REGION Network 7: CY26 interface H-shaftLoadingStopperCylinder4
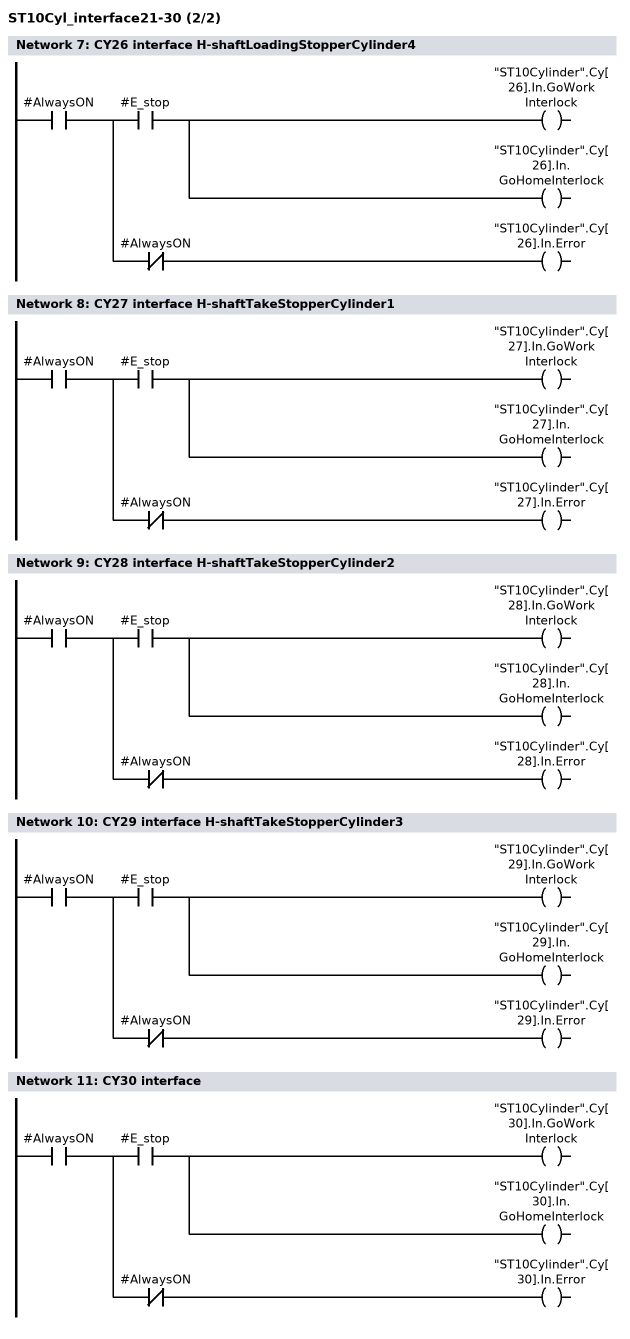
   RUNG wire#powerrail
      Contact( #AlwaysON )
      wire#w1
      Contact( #E_stop )
      wire#w2
      Coil( "ST10Cylinder".Cy[26].In.GoWorkInterlock )
   END_RUNG
   RUNG wire#w2
      Coil( "ST10Cylinder".Cy[26].In.GoHomeInterlock )
   END_RUNG
   RUNG wire#w1
      I_Contact( #AlwaysON )
      Coil( "ST10Cylinder".Cy[26].In.Error )
   END_RUNG
   // the same network as SCL:
   "ST10Cylinder".Cy[26].In.GoWorkInterlock := #AlwaysON AND #E_stop;
   "ST10Cylinder".Cy[26].In.GoHomeInterlock := #AlwaysON AND #E_stop;
   "ST10Cylinder".Cy[26].In.Error := #AlwaysON AND NOT #AlwaysON;
END_REGION

REGION Network 8: CY27 interface H-shaftTakeStopperCylinder1
   RUNG wire#powerrail
      Contact( #AlwaysON )
      wire#w1
      Contact( #E_stop )
      wire#w2
      Coil( "ST10Cylinder".Cy[27].In.GoWorkInterlock )
   END_RUNG
   RUNG wire#w2
      Coil( "ST10Cylinder".Cy[27].In.GoHomeInterlock )
   END_RUNG
   RUNG wire#w1
      I_Contact( #AlwaysON )
      Coil( "ST10Cylinder".Cy[27].In.Error )
   END_RUNG
   // the same network as SCL:
   "ST10Cylinder".Cy[27].In.GoWorkInterlock := #AlwaysON AND #E_stop;
   "ST10Cylinder".Cy[27].In.GoHomeInterlock := #AlwaysON AND #E_stop;
   "ST10Cylinder".Cy[27].In.Error := #AlwaysON AND NOT #AlwaysON;
END_REGION

REGION Network 9: CY28 interface H-shaftTakeStopperCylinder2
   RUNG wire#powerrail
      Contact( #AlwaysON )
      wire#w1
      Contact( #E_stop )
      wire#w2
      Coil( "ST10Cylinder".Cy[28].In.GoWorkInterlock )
   END_RUNG
   RUNG wire#w2
      Coil( "ST10Cylinder".Cy[28].In.GoHomeInterlock )
   END_RUNG
   RUNG wire#w1
      I_Contact( #AlwaysON )
      Coil( "ST10Cylinder".Cy[28].In.Error )
   END_RUNG
   // the same network as SCL:
   "ST10Cylinder".Cy[28].In.GoWorkInterlock := #AlwaysON AND #E_stop;
   "ST10Cylinder".Cy[28].In.GoHomeInterlock := #AlwaysON AND #E_stop;
   "ST10Cylinder".Cy[28].In.Error := #AlwaysON AND NOT #AlwaysON;
END_REGION

REGION Network 10: CY29 interface H-shaftTakeStopperCylinder3
   RUNG wire#powerrail
      Contact( #AlwaysON )
      wire#w1
      Contact( #E_stop )
      wire#w2
      Coil( "ST10Cylinder".Cy[29].In.GoWorkInterlock )
   END_RUNG
   RUNG wire#w2
      Coil( "ST10Cylinder".Cy[29].In.GoHomeInterlock )
   END_RUNG
   RUNG wire#w1
      I_Contact( #AlwaysON )
      Coil( "ST10Cylinder".Cy[29].In.Error )
   END_RUNG
   // the same network as SCL:
   "ST10Cylinder".Cy[29].In.GoWorkInterlock := #AlwaysON AND #E_stop;
   "ST10Cylinder".Cy[29].In.GoHomeInterlock := #AlwaysON AND #E_stop;
   "ST10Cylinder".Cy[29].In.Error := #AlwaysON AND NOT #AlwaysON;
END_REGION

REGION Network 11: CY30 interface
   RUNG wire#powerrail
      Contact( #AlwaysON )
      wire#w1
      Contact( #E_stop )
      wire#w2
      Coil( "ST10Cylinder".Cy[30].In.GoWorkInterlock )
   END_RUNG
   RUNG wire#w2
      Coil( "ST10Cylinder".Cy[30].In.GoHomeInterlock )
   END_RUNG
   RUNG wire#w1
      I_Contact( #AlwaysON )
      Coil( "ST10Cylinder".Cy[30].In.Error )
   END_RUNG
   // the same network as SCL:
   "ST10Cylinder".Cy[30].In.GoWorkInterlock := #AlwaysON AND #E_stop;
   "ST10Cylinder".Cy[30].In.GoHomeInterlock := #AlwaysON AND #E_stop;
   "ST10Cylinder".Cy[30].In.Error := #AlwaysON AND NOT #AlwaysON;
END_REGION
END_FUNCTION

FUNCTION "ST10Cyl_interface31-40" : Void   // FC1023, LAD
{ S7_Optimized_Access := 'FALSE' }
VERSION : 0.1
// stored: AutoNumber false, IsIECCheckEnabled false, SetENOAutomatically false, UDAEnableTagReadback false
   VAR_INPUT
      AlwaysON : Bool;
      E_stop : Bool;
   END_VAR
   VAR_TEMP
      tTest : Bool;
   END_VAR
BEGIN

REGION Network 1 (SCL): Cylinder 31-40 IO Interface (SCL)

   //Cylinder31 IO  J-magnetLiftingLiftingCylinder
   //Input
   "ST10Cylinder".Cy[31].In.WorkPositionSensor := "iJ-magnetLiftingLiftingCylinderInWP";
   "ST10Cylinder".Cy[31].In.HomePositionSensor := "iJ-magnetLiftingLiftingCylinderInHP";
   //Output
   "oJ-magnetLiftingLiftingCylinderToWP" := "ST10Cylinder".Cy[31].Out.GoWorkPosition;
   "oJ-magnetLiftingLiftingCylinderToHP" := "ST10Cylinder".Cy[31].Out.GoHomePosition;

   //Cylinder32 IO  J-magnetLiftingPalletLocationCylinder
   //Input
   "ST10Cylinder".Cy[32].In.WorkPositionSensor := "iJ-magnetLiftingPalletLocationCylinderInWP";
   "ST10Cylinder".Cy[32].In.HomePositionSensor := "iJ-magnetLiftingPalletLocationCylinderInHP";
   //Output
   "oJ-magnetLiftingPalletLocationCylinderToWP" := "ST10Cylinder".Cy[32].Out.GoWorkPosition;
   "oJ-magnetLiftingPalletLocationCylinderToHP" := "ST10Cylinder".Cy[32].Out.GoHomePosition;

   //Cylinder33 IO  J-magnetLoadingStopperCylinder1
   //Input
   "ST10Cylinder".Cy[33].In.WorkPositionSensor := "oJ-magnetLoadingStopperCylinder1_ToWP";
   "ST10Cylinder".Cy[33].In.HomePositionSensor := "oJ-magnetLoadingStopperCylinder1_ToHP";
   //Output
   "oJ-magnetLoadingStopperCylinder1_ToWP" := "ST10Cylinder".Cy[33].Out.GoWorkPosition;
   "oJ-magnetLoadingStopperCylinder1_ToHP" := "ST10Cylinder".Cy[33].Out.GoHomePosition;

   //Cylinder34 IO  J-magnetLoadingStopperCylinder2
   //Input
   "ST10Cylinder".Cy[34].In.WorkPositionSensor := "oJ-magnetLoadingStopperCylinder2_ToWP";
   "ST10Cylinder".Cy[34].In.HomePositionSensor := "oJ-magnetLoadingStopperCylinder2_ToHP";
   //Output
   "oJ-magnetLoadingStopperCylinder2_ToWP" := "ST10Cylinder".Cy[34].Out.GoWorkPosition;
   "oJ-magnetLoadingStopperCylinder2_ToHP" := "ST10Cylinder".Cy[34].Out.GoHomePosition;

   //Cylinder35 IO  J-magnetLoadingStopperCylinder3
   //Input
   "ST10Cylinder".Cy[35].In.WorkPositionSensor := "oJ-magnetLoadingStopperCylinder3_ToWP";
   "ST10Cylinder".Cy[35].In.HomePositionSensor := "oJ-magnetLoadingStopperCylinder3_ToHP";
   //Output
   "oJ-magnetLoadingStopperCylinder3_ToWP" := "ST10Cylinder".Cy[35].Out.GoWorkPosition;
   "oJ-magnetLoadingStopperCylinder3_ToHP" := "ST10Cylinder".Cy[35].Out.GoHomePosition;

   //Cylinder36 J-magnetLoadingStopperCylinder4
   //Input
   "ST10Cylinder".Cy[36].In.WorkPositionSensor := "oJ-magnetLoadingStopperCylinder4_ToWP";
   "ST10Cylinder".Cy[36].In.HomePositionSensor := "oJ-magnetLoadingStopperCylinder4_ToHP";
   //Output
   "oJ-magnetLoadingStopperCylinder4_ToWP" := "ST10Cylinder".Cy[36].Out.GoWorkPosition;
   "oJ-magnetLoadingStopperCylinder4_ToHP" := "ST10Cylinder".Cy[36].Out.GoHomePosition;

   //Cylinder37 J-magnetTakeStopperCylinder1
   //Input
   "ST10Cylinder".Cy[37].In.WorkPositionSensor := "oJ-magnetTakeStopperCylinder1_ToWP";
   "ST10Cylinder".Cy[37].In.HomePositionSensor := "oJ-magnetTakeStopperCylinder1_ToHP";
   //Output
   "oJ-magnetTakeStopperCylinder1_ToWP" := "ST10Cylinder".Cy[37].Out.GoWorkPosition;
   "oJ-magnetTakeStopperCylinder1_ToHP" := "ST10Cylinder".Cy[37].Out.GoHomePosition;

   //Cylinder38 J-magnetTakeStopperCylinder2
   //Input
   "ST10Cylinder".Cy[38].In.WorkPositionSensor := "oJ-magnetTakeStopperCylinder2_ToWP";
   "ST10Cylinder".Cy[38].In.HomePositionSensor := "oJ-magnetTakeStopperCylinder2_ToHP";
   //Output
   "oJ-magnetTakeStopperCylinder2_ToWP" := "ST10Cylinder".Cy[38].Out.GoWorkPosition;
   "oJ-magnetTakeStopperCylinder2_ToHP" := "ST10Cylinder".Cy[38].Out.GoHomePosition;

   //Cylinder39 J-magnetTakeStopperCylinder3
   //Input
   "ST10Cylinder".Cy[39].In.WorkPositionSensor := "oJ-magnetTakeStopperCylinder3_ToWP";
   "ST10Cylinder".Cy[39].In.HomePositionSensor := "oJ-magnetTakeStopperCylinder3_ToHP";
   //Output
   "oJ-magnetTakeStopperCylinder3_ToWP" := "ST10Cylinder".Cy[39].Out.GoWorkPosition;
   "oJ-magnetTakeStopperCylinder3_ToHP" := "ST10Cylinder".Cy[39].Out.GoHomePosition;

   (*
   //Cylinder40 J-magnetLoadingStopperCylinder4_2
   // //Input
   "ST10Cylinder".Cy[40].In.WorkPositionSensor := "oJ-magnetLoadingStopperCylinder4_2";
   "ST10Cylinder".Cy[40].In.HomePositionSensor := NOT "oJ-magnetLoadingStopperCylinder4_2";
   // //Output
   "oJ-magnetLoadingStopperCylinder4_2" := "ST10Cylinder".Cy[40].Out.GoWorkPosition;
   "Feeding washer  lift Cylinder ToHP" := "ST10Cylinder".Cy[40].Out.GoHomePosition;
   *)
END_REGION

REGION Network 2: CY31 interface J-magnetLiftingLiftingCylinder
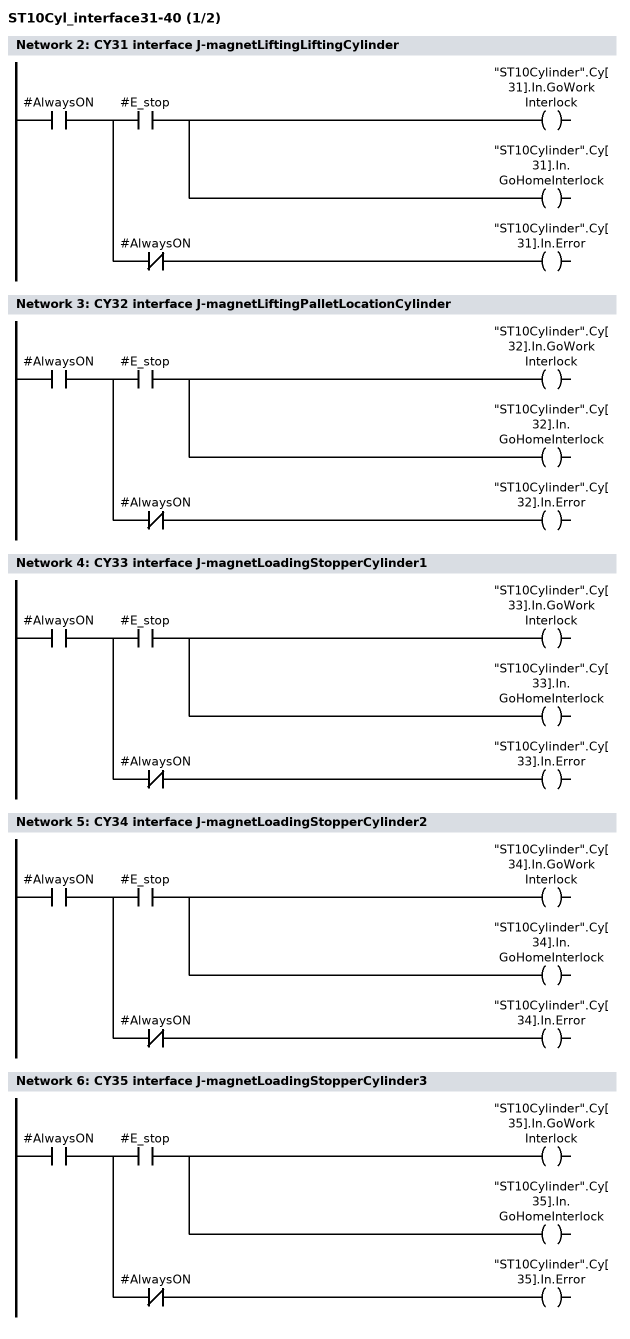
   RUNG wire#powerrail
      Contact( #AlwaysON )
      wire#w1
      Contact( #E_stop )
      wire#w2
      Coil( "ST10Cylinder".Cy[31].In.GoWorkInterlock )
   END_RUNG
   RUNG wire#w2
      Coil( "ST10Cylinder".Cy[31].In.GoHomeInterlock )
   END_RUNG
   RUNG wire#w1
      I_Contact( #AlwaysON )
      Coil( "ST10Cylinder".Cy[31].In.Error )
   END_RUNG
   // the same network as SCL:
   "ST10Cylinder".Cy[31].In.GoWorkInterlock := #AlwaysON AND #E_stop;
   "ST10Cylinder".Cy[31].In.GoHomeInterlock := #AlwaysON AND #E_stop;
   "ST10Cylinder".Cy[31].In.Error := #AlwaysON AND NOT #AlwaysON;
END_REGION

REGION Network 3: CY32 interface J-magnetLiftingPalletLocationCylinder
   RUNG wire#powerrail
      Contact( #AlwaysON )
      wire#w1
      Contact( #E_stop )
      wire#w2
      Coil( "ST10Cylinder".Cy[32].In.GoWorkInterlock )
   END_RUNG
   RUNG wire#w2
      Coil( "ST10Cylinder".Cy[32].In.GoHomeInterlock )
   END_RUNG
   RUNG wire#w1
      I_Contact( #AlwaysON )
      Coil( "ST10Cylinder".Cy[32].In.Error )
   END_RUNG
   // the same network as SCL:
   "ST10Cylinder".Cy[32].In.GoWorkInterlock := #AlwaysON AND #E_stop;
   "ST10Cylinder".Cy[32].In.GoHomeInterlock := #AlwaysON AND #E_stop;
   "ST10Cylinder".Cy[32].In.Error := #AlwaysON AND NOT #AlwaysON;
END_REGION

REGION Network 4: CY33 interface J-magnetLoadingStopperCylinder1
   RUNG wire#powerrail
      Contact( #AlwaysON )
      wire#w1
      Contact( #E_stop )
      wire#w2
      Coil( "ST10Cylinder".Cy[33].In.GoWorkInterlock )
   END_RUNG
   RUNG wire#w2
      Coil( "ST10Cylinder".Cy[33].In.GoHomeInterlock )
   END_RUNG
   RUNG wire#w1
      I_Contact( #AlwaysON )
      Coil( "ST10Cylinder".Cy[33].In.Error )
   END_RUNG
   // the same network as SCL:
   "ST10Cylinder".Cy[33].In.GoWorkInterlock := #AlwaysON AND #E_stop;
   "ST10Cylinder".Cy[33].In.GoHomeInterlock := #AlwaysON AND #E_stop;
   "ST10Cylinder".Cy[33].In.Error := #AlwaysON AND NOT #AlwaysON;
END_REGION

REGION Network 5: CY34 interface J-magnetLoadingStopperCylinder2
   RUNG wire#powerrail
      Contact( #AlwaysON )
      wire#w1
      Contact( #E_stop )
      wire#w2
      Coil( "ST10Cylinder".Cy[34].In.GoWorkInterlock )
   END_RUNG
   RUNG wire#w2
      Coil( "ST10Cylinder".Cy[34].In.GoHomeInterlock )
   END_RUNG
   RUNG wire#w1
      I_Contact( #AlwaysON )
      Coil( "ST10Cylinder".Cy[34].In.Error )
   END_RUNG
   // the same network as SCL:
   "ST10Cylinder".Cy[34].In.GoWorkInterlock := #AlwaysON AND #E_stop;
   "ST10Cylinder".Cy[34].In.GoHomeInterlock := #AlwaysON AND #E_stop;
   "ST10Cylinder".Cy[34].In.Error := #AlwaysON AND NOT #AlwaysON;
END_REGION

REGION Network 6: CY35 interface J-magnetLoadingStopperCylinder3
   RUNG wire#powerrail
      Contact( #AlwaysON )
      wire#w1
      Contact( #E_stop )
      wire#w2
      Coil( "ST10Cylinder".Cy[35].In.GoWorkInterlock )
   END_RUNG
   RUNG wire#w2
      Coil( "ST10Cylinder".Cy[35].In.GoHomeInterlock )
   END_RUNG
   RUNG wire#w1
      I_Contact( #AlwaysON )
      Coil( "ST10Cylinder".Cy[35].In.Error )
   END_RUNG
   // the same network as SCL:
   "ST10Cylinder".Cy[35].In.GoWorkInterlock := #AlwaysON AND #E_stop;
   "ST10Cylinder".Cy[35].In.GoHomeInterlock := #AlwaysON AND #E_stop;
   "ST10Cylinder".Cy[35].In.Error := #AlwaysON AND NOT #AlwaysON;
END_REGION

REGION Network 7: CY36 interface J-magnetLoadingStopperCylinder4
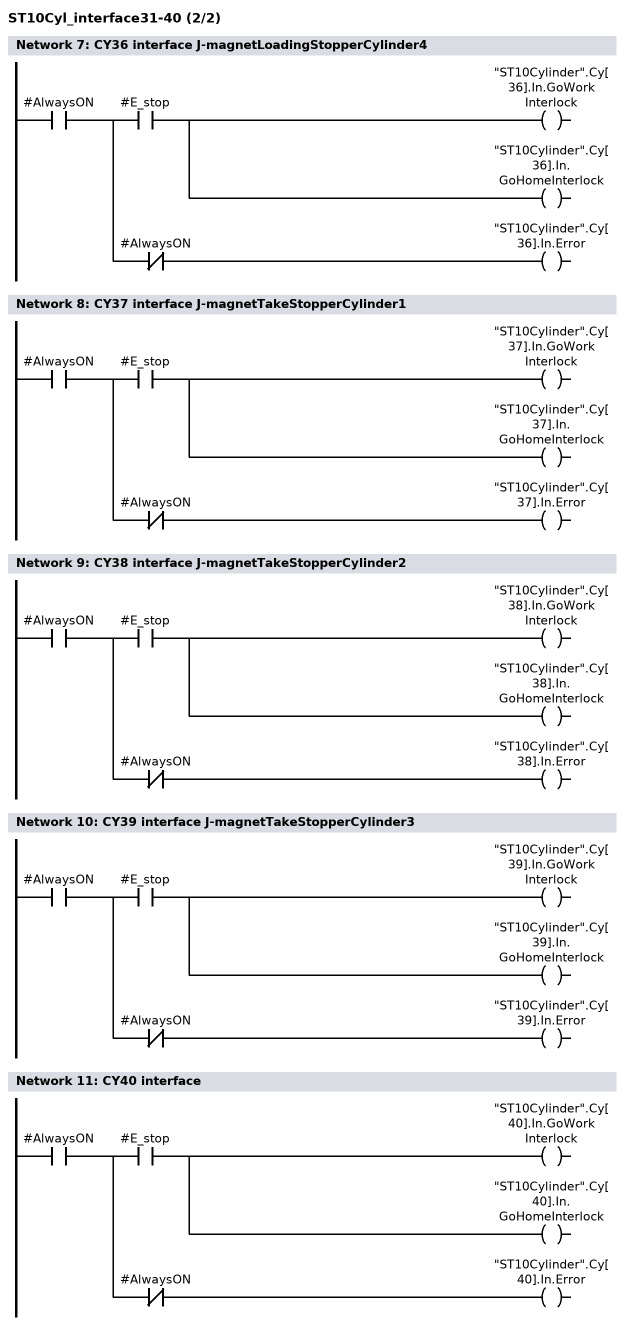
   RUNG wire#powerrail
      Contact( #AlwaysON )
      wire#w1
      Contact( #E_stop )
      wire#w2
      Coil( "ST10Cylinder".Cy[36].In.GoWorkInterlock )
   END_RUNG
   RUNG wire#w2
      Coil( "ST10Cylinder".Cy[36].In.GoHomeInterlock )
   END_RUNG
   RUNG wire#w1
      I_Contact( #AlwaysON )
      Coil( "ST10Cylinder".Cy[36].In.Error )
   END_RUNG
   // the same network as SCL:
   "ST10Cylinder".Cy[36].In.GoWorkInterlock := #AlwaysON AND #E_stop;
   "ST10Cylinder".Cy[36].In.GoHomeInterlock := #AlwaysON AND #E_stop;
   "ST10Cylinder".Cy[36].In.Error := #AlwaysON AND NOT #AlwaysON;
END_REGION

REGION Network 8: CY37 interface J-magnetTakeStopperCylinder1
   RUNG wire#powerrail
      Contact( #AlwaysON )
      wire#w1
      Contact( #E_stop )
      wire#w2
      Coil( "ST10Cylinder".Cy[37].In.GoWorkInterlock )
   END_RUNG
   RUNG wire#w2
      Coil( "ST10Cylinder".Cy[37].In.GoHomeInterlock )
   END_RUNG
   RUNG wire#w1
      I_Contact( #AlwaysON )
      Coil( "ST10Cylinder".Cy[37].In.Error )
   END_RUNG
   // the same network as SCL:
   "ST10Cylinder".Cy[37].In.GoWorkInterlock := #AlwaysON AND #E_stop;
   "ST10Cylinder".Cy[37].In.GoHomeInterlock := #AlwaysON AND #E_stop;
   "ST10Cylinder".Cy[37].In.Error := #AlwaysON AND NOT #AlwaysON;
END_REGION

REGION Network 9: CY38 interface J-magnetTakeStopperCylinder2
   RUNG wire#powerrail
      Contact( #AlwaysON )
      wire#w1
      Contact( #E_stop )
      wire#w2
      Coil( "ST10Cylinder".Cy[38].In.GoWorkInterlock )
   END_RUNG
   RUNG wire#w2
      Coil( "ST10Cylinder".Cy[38].In.GoHomeInterlock )
   END_RUNG
   RUNG wire#w1
      I_Contact( #AlwaysON )
      Coil( "ST10Cylinder".Cy[38].In.Error )
   END_RUNG
   // the same network as SCL:
   "ST10Cylinder".Cy[38].In.GoWorkInterlock := #AlwaysON AND #E_stop;
   "ST10Cylinder".Cy[38].In.GoHomeInterlock := #AlwaysON AND #E_stop;
   "ST10Cylinder".Cy[38].In.Error := #AlwaysON AND NOT #AlwaysON;
END_REGION

REGION Network 10: CY39 interface J-magnetTakeStopperCylinder3
   RUNG wire#powerrail
      Contact( #AlwaysON )
      wire#w1
      Contact( #E_stop )
      wire#w2
      Coil( "ST10Cylinder".Cy[39].In.GoWorkInterlock )
   END_RUNG
   RUNG wire#w2
      Coil( "ST10Cylinder".Cy[39].In.GoHomeInterlock )
   END_RUNG
   RUNG wire#w1
      I_Contact( #AlwaysON )
      Coil( "ST10Cylinder".Cy[39].In.Error )
   END_RUNG
   // the same network as SCL:
   "ST10Cylinder".Cy[39].In.GoWorkInterlock := #AlwaysON AND #E_stop;
   "ST10Cylinder".Cy[39].In.GoHomeInterlock := #AlwaysON AND #E_stop;
   "ST10Cylinder".Cy[39].In.Error := #AlwaysON AND NOT #AlwaysON;
END_REGION

REGION Network 11: CY40 interface
   RUNG wire#powerrail
      Contact( #AlwaysON )
      wire#w1
      Contact( #E_stop )
      wire#w2
      Coil( "ST10Cylinder".Cy[40].In.GoWorkInterlock )
   END_RUNG
   RUNG wire#w2
      Coil( "ST10Cylinder".Cy[40].In.GoHomeInterlock )
   END_RUNG
   RUNG wire#w1
      I_Contact( #AlwaysON )
      Coil( "ST10Cylinder".Cy[40].In.Error )
   END_RUNG
   // the same network as SCL:
   "ST10Cylinder".Cy[40].In.GoWorkInterlock := #AlwaysON AND #E_stop;
   "ST10Cylinder".Cy[40].In.GoHomeInterlock := #AlwaysON AND #E_stop;
   "ST10Cylinder".Cy[40].In.Error := #AlwaysON AND NOT #AlwaysON;
END_REGION
END_FUNCTION

FUNCTION "ST10Cyl_interface41-50" : Void   // FC1024, LAD
{ S7_Optimized_Access := 'FALSE' }
// stored: AutoNumber false, SetENOAutomatically false
   VAR_INPUT
      AlwaysON : Bool;
      E_stop : Bool;
   END_VAR
   VAR_TEMP
      tTest : Bool;
   END_VAR
BEGIN

REGION Network 1 (SCL): Cylinder 41-50 IO Interface (SCL)
   //Cylinder41 IO  K-reserveLifting3LiftingCylinder
   //Input
   "ST10Cylinder".Cy[41].In.WorkPositionSensor := "iK-reserveLifting3LiftingCylinderInWP";
   "ST10Cylinder".Cy[41].In.HomePositionSensor := "iK-reserveLifting3LiftingCylinderInHP";
   //Output
   "oK-reserveLifting3LiftingCylinderToWP" := "ST10Cylinder".Cy[41].Out.GoWorkPosition;
   "oK-reserveLifting3LiftingCylinderToHP" := "ST10Cylinder".Cy[41].Out.GoHomePosition;

   //Cylinder42 IO  K-reserveLifting3PalletLocationCylinder
   //Input
   "ST10Cylinder".Cy[42].In.WorkPositionSensor := "iK-reserveLifting3PalletLocationCylinderInWP";
   "ST10Cylinder".Cy[42].In.HomePositionSensor := "iK-reserveLifting3PalletLocationCylinderInHP";
   //Output
   "oK-reserveLifting3PalletLocationCylinderToWP" := "ST10Cylinder".Cy[42].Out.GoWorkPosition;
   "oK-reserveLifting3PalletLocationCylinderToHP" := "ST10Cylinder".Cy[42].Out.GoHomePosition;

   //Cylinder43 IO  K-reserveLoadingStopperCylinder1
   //Input
   "ST10Cylinder".Cy[43].In.WorkPositionSensor := "oK-reserveLoadingStopperCylinder1_ToWP";
   "ST10Cylinder".Cy[43].In.HomePositionSensor := "oK-reserveLoadingStopperCylinder1_ToHP";
   //Output
   "oK-reserveLoadingStopperCylinder1_ToWP" := "ST10Cylinder".Cy[43].Out.GoWorkPosition;
   "oK-reserveLoadingStopperCylinder1_ToHP" := "ST10Cylinder".Cy[43].Out.GoHomePosition;

   //Cylinder44 IO  K-reserveLoadingStopperCylinder2
   //Input
   "ST10Cylinder".Cy[44].In.WorkPositionSensor := "oK-reserveLoadingStopperCylinder2_ToWP";
   "ST10Cylinder".Cy[44].In.HomePositionSensor := "oK-reserveLoadingStopperCylinder2_ToHP";
   //Output
   "oK-reserveLoadingStopperCylinder2_ToWP" := "ST10Cylinder".Cy[44].Out.GoWorkPosition;
   "oK-reserveLoadingStopperCylinder2_ToHP" := "ST10Cylinder".Cy[44].Out.GoHomePosition;

   //Cylinder45 IO  K-reserveLoadingStopperCylinder3
   //Input
   "ST10Cylinder".Cy[45].In.WorkPositionSensor := "oK-reserveLoadingStopperCylinder3_ToWP";
   "ST10Cylinder".Cy[45].In.HomePositionSensor := "oK-reserveLoadingStopperCylinder3_ToHP";
   //Output
   "oK-reserveLoadingStopperCylinder3_ToWP" := "ST10Cylinder".Cy[45].Out.GoWorkPosition;
   "oK-reserveLoadingStopperCylinder3_ToHP" := "ST10Cylinder".Cy[45].Out.GoHomePosition;

   //Cylinder46 K-reserveLoadingStopperCylinder4
   //Input
   "ST10Cylinder".Cy[46].In.WorkPositionSensor := "oK-reserveLoadingStopperCylinder4_ToWP";
   "ST10Cylinder".Cy[46].In.HomePositionSensor := "oK-reserveLoadingStopperCylinder4_ToHP";
   //Output
   "oK-reserveLoadingStopperCylinder4_ToWP" := "ST10Cylinder".Cy[46].Out.GoWorkPosition;
   "oK-reserveLoadingStopperCylinder4_ToHP" := "ST10Cylinder".Cy[46].Out.GoHomePosition;

   //Cylinder47 K-reserveTakeStopperCylinder1
   //Input
   "ST10Cylinder".Cy[47].In.WorkPositionSensor := "oK-reserveTakeStopperCylinder1_ToWP";
   "ST10Cylinder".Cy[47].In.HomePositionSensor := "oK-reserveTakeStopperCylinder1_ToHP";
   //Output
   "oK-reserveTakeStopperCylinder1_ToWP" := "ST10Cylinder".Cy[47].Out.GoWorkPosition;
   "oK-reserveTakeStopperCylinder1_ToHP" := "ST10Cylinder".Cy[47].Out.GoHomePosition;

   //Cylinder48 K-reserveTakeStopperCylinder2
   //Input
   "ST10Cylinder".Cy[48].In.WorkPositionSensor := "oK-reserveTakeStopperCylinder2_ToWP";
   "ST10Cylinder".Cy[48].In.HomePositionSensor := "oK-reserveTakeStopperCylinder2_ToHP";
   //Output
   "oK-reserveTakeStopperCylinder2_ToWP" := "ST10Cylinder".Cy[48].Out.GoWorkPosition;
   "oK-reserveTakeStopperCylinder2_ToHP" := "ST10Cylinder".Cy[48].Out.GoHomePosition;

   //Cylinder49 K-reserveTakeStopperCylinder3
   //Input
   "ST10Cylinder".Cy[49].In.WorkPositionSensor := "oK-reserveTakeStopperCylinder3_ToWP";
   "ST10Cylinder".Cy[49].In.HomePositionSensor := "oK-reserveTakeStopperCylinder3_ToHP";
   //Output
   "oK-reserveTakeStopperCylinder3_ToWP" := "ST10Cylinder".Cy[49].Out.GoWorkPosition;
   "oK-reserveTakeStopperCylinder3_ToHP" := "ST10Cylinder".Cy[49].Out.GoHomePosition;

   (*
   //Cylinder50 K-reserveLoadingStopperCylinder4_2
   // //Input
   "ST10Cylinder".Cy[50].In.WorkPositionSensor := "oK-reserveLoadingStopperCylinder4_2";
   "ST10Cylinder".Cy[50].In.HomePositionSensor := NOT "oK-reserveLoadingStopperCylinder4_2";
   // //Output
   "oK-reserveLoadingStopperCylinder4_2" := "ST10Cylinder".Cy[50].Out.GoWorkPosition;
   // "Feeding washer  lift Cylinder ToHP" := "ST10Cylinder".Cy[50].Out.GoHomePosition;
   *)
END_REGION

REGION Network 2: CY41 interface K-reserveLifting3LiftingCylinder
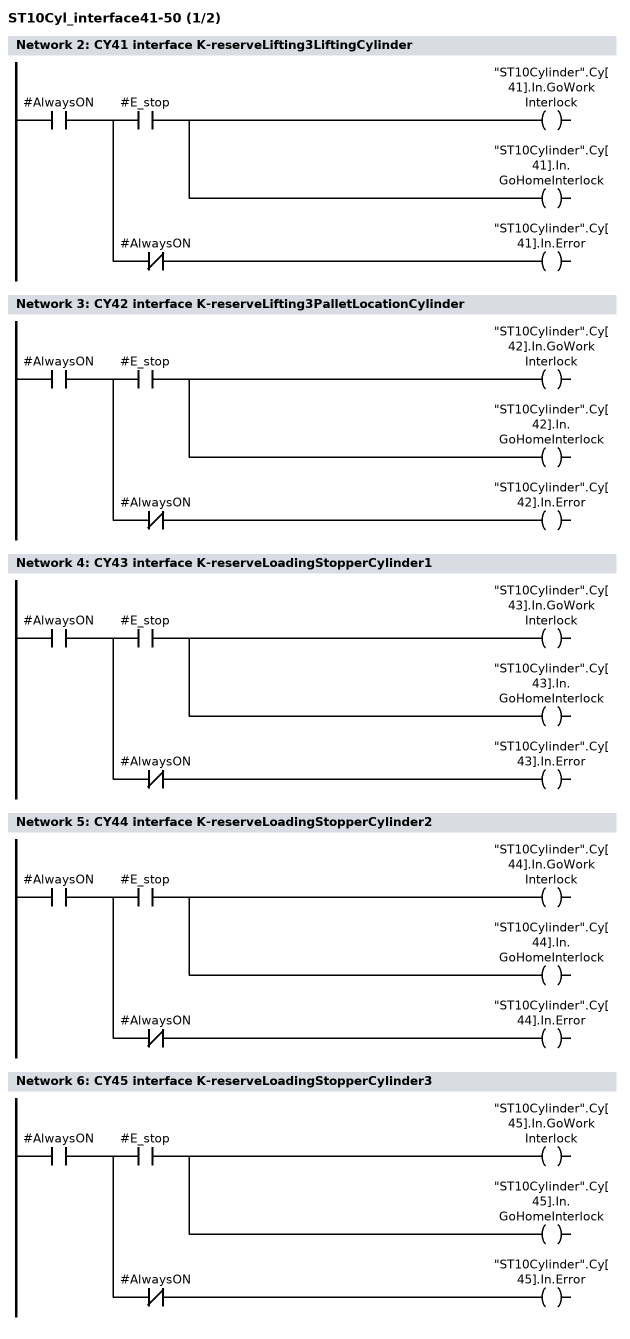
   RUNG wire#powerrail
      Contact( #AlwaysON )
      wire#w1
      Contact( #E_stop )
      wire#w2
      Coil( "ST10Cylinder".Cy[41].In.GoWorkInterlock )
   END_RUNG
   RUNG wire#w2
      Coil( "ST10Cylinder".Cy[41].In.GoHomeInterlock )
   END_RUNG
   RUNG wire#w1
      I_Contact( #AlwaysON )
      Coil( "ST10Cylinder".Cy[41].In.Error )
   END_RUNG
   // the same network as SCL:
   "ST10Cylinder".Cy[41].In.GoWorkInterlock := #AlwaysON AND #E_stop;
   "ST10Cylinder".Cy[41].In.GoHomeInterlock := #AlwaysON AND #E_stop;
   "ST10Cylinder".Cy[41].In.Error := #AlwaysON AND NOT #AlwaysON;
END_REGION

REGION Network 3: CY42 interface K-reserveLifting3PalletLocationCylinder
   RUNG wire#powerrail
      Contact( #AlwaysON )
      wire#w1
      Contact( #E_stop )
      wire#w2
      Coil( "ST10Cylinder".Cy[42].In.GoWorkInterlock )
   END_RUNG
   RUNG wire#w2
      Coil( "ST10Cylinder".Cy[42].In.GoHomeInterlock )
   END_RUNG
   RUNG wire#w1
      I_Contact( #AlwaysON )
      Coil( "ST10Cylinder".Cy[42].In.Error )
   END_RUNG
   // the same network as SCL:
   "ST10Cylinder".Cy[42].In.GoWorkInterlock := #AlwaysON AND #E_stop;
   "ST10Cylinder".Cy[42].In.GoHomeInterlock := #AlwaysON AND #E_stop;
   "ST10Cylinder".Cy[42].In.Error := #AlwaysON AND NOT #AlwaysON;
END_REGION

REGION Network 4: CY43 interface K-reserveLoadingStopperCylinder1
   RUNG wire#powerrail
      Contact( #AlwaysON )
      wire#w1
      Contact( #E_stop )
      wire#w2
      Coil( "ST10Cylinder".Cy[43].In.GoWorkInterlock )
   END_RUNG
   RUNG wire#w2
      Coil( "ST10Cylinder".Cy[43].In.GoHomeInterlock )
   END_RUNG
   RUNG wire#w1
      I_Contact( #AlwaysON )
      Coil( "ST10Cylinder".Cy[43].In.Error )
   END_RUNG
   // the same network as SCL:
   "ST10Cylinder".Cy[43].In.GoWorkInterlock := #AlwaysON AND #E_stop;
   "ST10Cylinder".Cy[43].In.GoHomeInterlock := #AlwaysON AND #E_stop;
   "ST10Cylinder".Cy[43].In.Error := #AlwaysON AND NOT #AlwaysON;
END_REGION

REGION Network 5: CY44 interface K-reserveLoadingStopperCylinder2
   RUNG wire#powerrail
      Contact( #AlwaysON )
      wire#w1
      Contact( #E_stop )
      wire#w2
      Coil( "ST10Cylinder".Cy[44].In.GoWorkInterlock )
   END_RUNG
   RUNG wire#w2
      Coil( "ST10Cylinder".Cy[44].In.GoHomeInterlock )
   END_RUNG
   RUNG wire#w1
      I_Contact( #AlwaysON )
      Coil( "ST10Cylinder".Cy[44].In.Error )
   END_RUNG
   // the same network as SCL:
   "ST10Cylinder".Cy[44].In.GoWorkInterlock := #AlwaysON AND #E_stop;
   "ST10Cylinder".Cy[44].In.GoHomeInterlock := #AlwaysON AND #E_stop;
   "ST10Cylinder".Cy[44].In.Error := #AlwaysON AND NOT #AlwaysON;
END_REGION

REGION Network 6: CY45 interface K-reserveLoadingStopperCylinder3
   RUNG wire#powerrail
      Contact( #AlwaysON )
      wire#w1
      Contact( #E_stop )
      wire#w2
      Coil( "ST10Cylinder".Cy[45].In.GoWorkInterlock )
   END_RUNG
   RUNG wire#w2
      Coil( "ST10Cylinder".Cy[45].In.GoHomeInterlock )
   END_RUNG
   RUNG wire#w1
      I_Contact( #AlwaysON )
      Coil( "ST10Cylinder".Cy[45].In.Error )
   END_RUNG
   // the same network as SCL:
   "ST10Cylinder".Cy[45].In.GoWorkInterlock := #AlwaysON AND #E_stop;
   "ST10Cylinder".Cy[45].In.GoHomeInterlock := #AlwaysON AND #E_stop;
   "ST10Cylinder".Cy[45].In.Error := #AlwaysON AND NOT #AlwaysON;
END_REGION

REGION Network 7: CY46 interface K-reserveLoadingStopperCylinder4
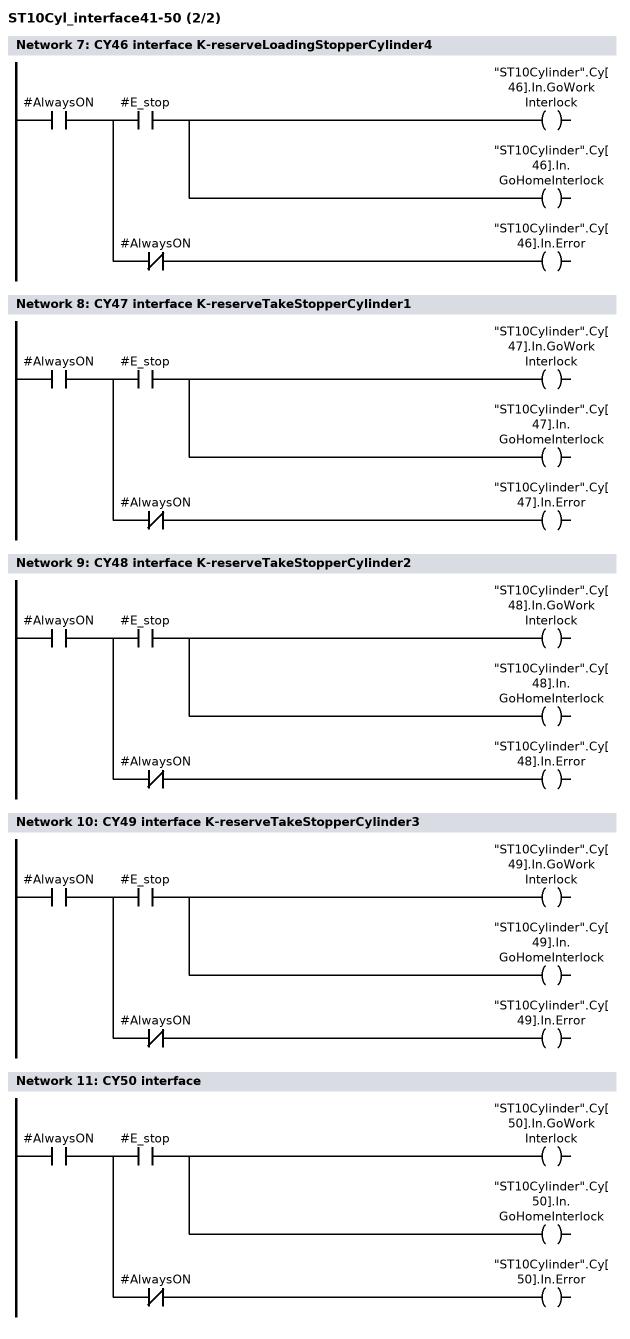
   RUNG wire#powerrail
      Contact( #AlwaysON )
      wire#w1
      Contact( #E_stop )
      wire#w2
      Coil( "ST10Cylinder".Cy[46].In.GoWorkInterlock )
   END_RUNG
   RUNG wire#w2
      Coil( "ST10Cylinder".Cy[46].In.GoHomeInterlock )
   END_RUNG
   RUNG wire#w1
      I_Contact( #AlwaysON )
      Coil( "ST10Cylinder".Cy[46].In.Error )
   END_RUNG
   // the same network as SCL:
   "ST10Cylinder".Cy[46].In.GoWorkInterlock := #AlwaysON AND #E_stop;
   "ST10Cylinder".Cy[46].In.GoHomeInterlock := #AlwaysON AND #E_stop;
   "ST10Cylinder".Cy[46].In.Error := #AlwaysON AND NOT #AlwaysON;
END_REGION

REGION Network 8: CY47 interface K-reserveTakeStopperCylinder1
   RUNG wire#powerrail
      Contact( #AlwaysON )
      wire#w1
      Contact( #E_stop )
      wire#w2
      Coil( "ST10Cylinder".Cy[47].In.GoWorkInterlock )
   END_RUNG
   RUNG wire#w2
      Coil( "ST10Cylinder".Cy[47].In.GoHomeInterlock )
   END_RUNG
   RUNG wire#w1
      I_Contact( #AlwaysON )
      Coil( "ST10Cylinder".Cy[47].In.Error )
   END_RUNG
   // the same network as SCL:
   "ST10Cylinder".Cy[47].In.GoWorkInterlock := #AlwaysON AND #E_stop;
   "ST10Cylinder".Cy[47].In.GoHomeInterlock := #AlwaysON AND #E_stop;
   "ST10Cylinder".Cy[47].In.Error := #AlwaysON AND NOT #AlwaysON;
END_REGION

REGION Network 9: CY48 interface K-reserveTakeStopperCylinder2
   RUNG wire#powerrail
      Contact( #AlwaysON )
      wire#w1
      Contact( #E_stop )
      wire#w2
      Coil( "ST10Cylinder".Cy[48].In.GoWorkInterlock )
   END_RUNG
   RUNG wire#w2
      Coil( "ST10Cylinder".Cy[48].In.GoHomeInterlock )
   END_RUNG
   RUNG wire#w1
      I_Contact( #AlwaysON )
      Coil( "ST10Cylinder".Cy[48].In.Error )
   END_RUNG
   // the same network as SCL:
   "ST10Cylinder".Cy[48].In.GoWorkInterlock := #AlwaysON AND #E_stop;
   "ST10Cylinder".Cy[48].In.GoHomeInterlock := #AlwaysON AND #E_stop;
   "ST10Cylinder".Cy[48].In.Error := #AlwaysON AND NOT #AlwaysON;
END_REGION

REGION Network 10: CY49 interface K-reserveTakeStopperCylinder3
   RUNG wire#powerrail
      Contact( #AlwaysON )
      wire#w1
      Contact( #E_stop )
      wire#w2
      Coil( "ST10Cylinder".Cy[49].In.GoWorkInterlock )
   END_RUNG
   RUNG wire#w2
      Coil( "ST10Cylinder".Cy[49].In.GoHomeInterlock )
   END_RUNG
   RUNG wire#w1
      I_Contact( #AlwaysON )
      Coil( "ST10Cylinder".Cy[49].In.Error )
   END_RUNG
   // the same network as SCL:
   "ST10Cylinder".Cy[49].In.GoWorkInterlock := #AlwaysON AND #E_stop;
   "ST10Cylinder".Cy[49].In.GoHomeInterlock := #AlwaysON AND #E_stop;
   "ST10Cylinder".Cy[49].In.Error := #AlwaysON AND NOT #AlwaysON;
END_REGION

REGION Network 11: CY50 interface
   RUNG wire#powerrail
      Contact( #AlwaysON )
      wire#w1
      Contact( #E_stop )
      wire#w2
      Coil( "ST10Cylinder".Cy[50].In.GoWorkInterlock )
   END_RUNG
   RUNG wire#w2
      Coil( "ST10Cylinder".Cy[50].In.GoHomeInterlock )
   END_RUNG
   RUNG wire#w1
      I_Contact( #AlwaysON )
      Coil( "ST10Cylinder".Cy[50].In.Error )
   END_RUNG
   // the same network as SCL:
   "ST10Cylinder".Cy[50].In.GoWorkInterlock := #AlwaysON AND #E_stop;
   "ST10Cylinder".Cy[50].In.GoHomeInterlock := #AlwaysON AND #E_stop;
   "ST10Cylinder".Cy[50].In.Error := #AlwaysON AND NOT #AlwaysON;
END_REGION
END_FUNCTION

FUNCTION "ST10Cyl_interface51-60" : Void   // FC1025, LAD
{ S7_Optimized_Access := 'FALSE' }
VERSION : 0.1
// stored: AutoNumber false, IsIECCheckEnabled false, SetENOAutomatically false, UDAEnableTagReadback false
   VAR_INPUT
      AlwaysON : Bool;
      E_stop : Bool;
   END_VAR
   VAR_TEMP
      tTest : Bool;
   END_VAR
   VAR_TEMP   // added for the SCL form of the ladder/FBD networks
      _w1 : Bool;
   END_VAR
BEGIN

REGION Network 1 (SCL): Cylinder 51-60 IO Interface (SCL)

   //Cylinder51 IO  L-UnloadingTransCylinder
   //Input
   "ST10Cylinder".Cy[51].In.WorkPositionSensor := "iL-UnloadingTransCylinderInWP";
   "ST10Cylinder".Cy[51].In.HomePositionSensor := "iL-UnloadingTransCylinderInHP";
   //Output
   "oL-UnloadingTransCylinderToWP" := "ST10Cylinder".Cy[51].Out.GoWorkPosition;
   "oL-UnloadingTransCylinderToHP" := "ST10Cylinder".Cy[51].Out.GoHomePosition;

   //Cylinder52 IO  L-UnloadingTransPalletLocationCylinder
   //Input
   "ST10Cylinder".Cy[52].In.WorkPositionSensor := "iL-UnloadingTransPalletLocationCylinderInWP";
   "ST10Cylinder".Cy[52].In.HomePositionSensor := "iL-UnloadingTransPalletLocationCylinderInHP";
   //Output
   "oL-UnloadingTransPalletLocationCylinderToWP" := "ST10Cylinder".Cy[52].Out.GoWorkPosition;
   "oL-UnloadingTransPalletLocationCylinderToHP" := "ST10Cylinder".Cy[52].Out.GoHomePosition;

   //Cylinder53 IO  L-UnloadingStopperCylinder1
   //Input
   "ST10Cylinder".Cy[53].In.WorkPositionSensor := "oL-UnloadingStopperCylinder1_ToWP";
   "ST10Cylinder".Cy[53].In.HomePositionSensor := "oL-UnloadingStopperCylinder1_ToHP";
   //Output
   "oL-UnloadingStopperCylinder1_ToWP" := "ST10Cylinder".Cy[53].Out.GoWorkPosition;
   "oL-UnloadingStopperCylinder1_ToHP" := "ST10Cylinder".Cy[53].Out.GoHomePosition;

   //Cylinder54 IO  L-UnloadingStopperCylinder2
   //Input
   "ST10Cylinder".Cy[54].In.WorkPositionSensor := "oL-UnloadingStopperCylinder2_ToWP";
   "ST10Cylinder".Cy[54].In.HomePositionSensor := "oL-UnloadingStopperCylinder2_ToHP";
   //Output
   "oL-UnloadingStopperCylinder2_ToWP" := "ST10Cylinder".Cy[54].Out.GoWorkPosition;
   "oL-UnloadingStopperCylinder2_ToHP" := "ST10Cylinder".Cy[54].Out.GoHomePosition;

   //Cylinder55 IO  L-UnloadingStopperCylinder3
   //Input
   "ST10Cylinder".Cy[55].In.WorkPositionSensor := "oL-UnloadingStopperCylinder3_ToWP";
   "ST10Cylinder".Cy[55].In.HomePositionSensor := "oL-UnloadingStopperCylinder3_ToHP";
   //Output
   "oL-UnloadingStopperCylinder3_ToWP" := "ST10Cylinder".Cy[55].Out.GoWorkPosition;
   "oL-UnloadingStopperCylinder3_ToHP" := "ST10Cylinder".Cy[55].Out.GoHomePosition;

   (*
   //Cylinder56  L-UnloadingStopperCylinder2_2
   //Input
   "ST10Cylinder".Cy[56].In.WorkPositionSensor := "oL-UnloadingStopperCylinder2_2";
   "ST10Cylinder".Cy[56].In.HomePositionSensor := NOT "oL-UnloadingStopperCylinder2_2";
   //Output
   "oL-UnloadingStopperCylinder2_2" := "ST10Cylinder".Cy[56].Out.GoWorkPosition;
   //"oI-0080TrayLoadingTraySupportCylinder1ToHP" := "ST10Cylinder".Cy[56].Out.GoHomePosition;

   //Cylinder57 L-UnloadingStopperCylinder3_1
   //Input
   "ST10Cylinder".Cy[57].In.WorkPositionSensor := "oL-UnloadingStopperCylinder3_1";
   "ST10Cylinder".Cy[57].In.HomePositionSensor := NOT "oL-UnloadingStopperCylinder3_1";
   //Output
   "oL-UnloadingStopperCylinder3_1" := "ST10Cylinder".Cy[57].Out.GoWorkPosition;
   //"oI-0070TrayLoadingTraySupportCylinder8ToHP" := "ST10Cylinder".Cy[57].Out.GoHomePosition;

   //Cylinder58 L-UnloadingStopperCylinder3_2
   //Input
   "ST10Cylinder".Cy[58].In.WorkPositionSensor := "oL-UnloadingStopperCylinder3_2";
   "ST10Cylinder".Cy[58].In.HomePositionSensor := NOT "oL-UnloadingStopperCylinder3_2";
   //Output
   "oL-UnloadingStopperCylinder3_2" := "ST10Cylinder".Cy[58].Out.GoWorkPosition;
   //"oI-0080TrayLoadingTrayLocationCylinderToHP" := "ST10Cylinder".Cy[58].Out.GoHomePosition;
   //

   *)
END_REGION

REGION Network 2: CY51 interface L-UnloadingTransCylinder
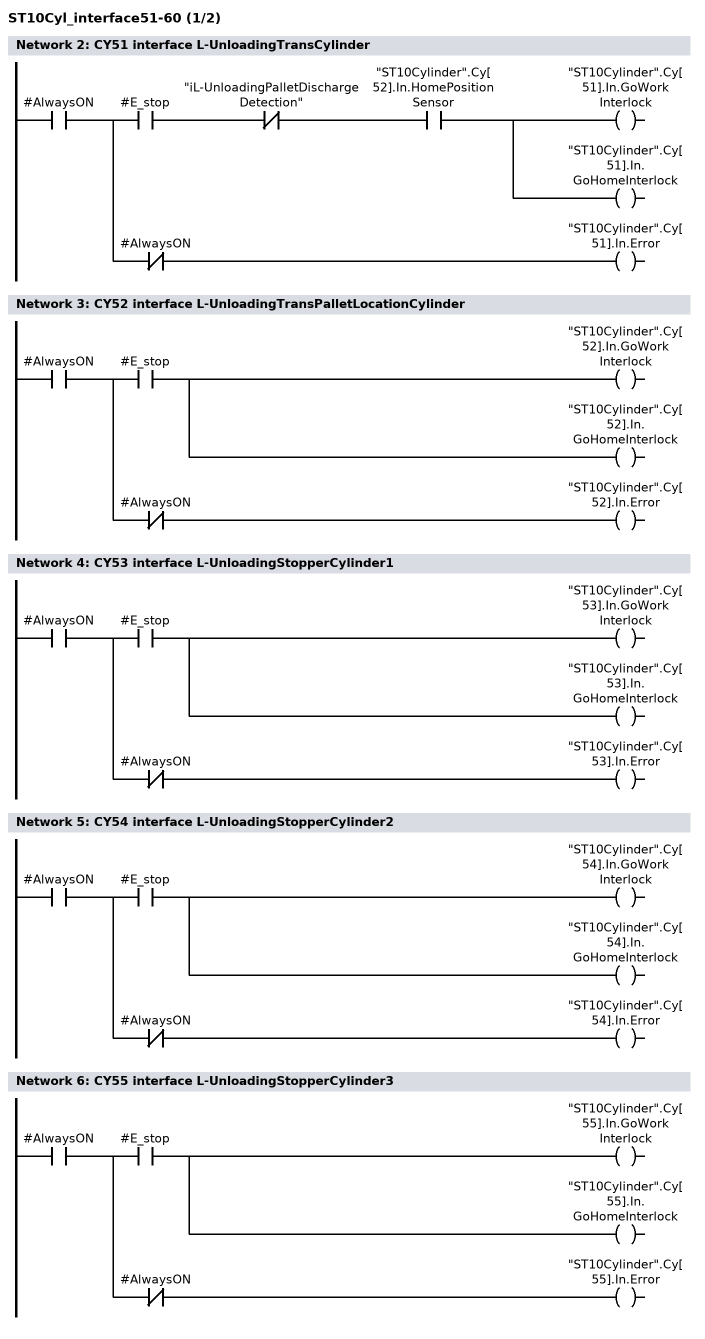
   RUNG wire#powerrail
      Contact( #AlwaysON )
      wire#w1
      Contact( #E_stop )
      I_Contact( "iL-UnloadingPalletDischargeDetection" )
      Contact( "ST10Cylinder".Cy[52].In.HomePositionSensor )
      wire#w2
      Coil( "ST10Cylinder".Cy[51].In.GoWorkInterlock )
   END_RUNG
   RUNG wire#w2
      Coil( "ST10Cylinder".Cy[51].In.GoHomeInterlock )
   END_RUNG
   RUNG wire#w1
      I_Contact( #AlwaysON )
      Coil( "ST10Cylinder".Cy[51].In.Error )
   END_RUNG
   // the same network as SCL:
   #_w1 := #AlwaysON AND #E_stop AND NOT "iL-UnloadingPalletDischargeDetection" AND "ST10Cylinder".Cy[52].In.HomePositionSensor;
   "ST10Cylinder".Cy[51].In.GoWorkInterlock := #AlwaysON AND #E_stop AND NOT "iL-UnloadingPalletDischargeDetection" AND "ST10Cylinder".Cy[52].In.HomePositionSensor;
   "ST10Cylinder".Cy[51].In.GoHomeInterlock := #_w1;
   "ST10Cylinder".Cy[51].In.Error := #AlwaysON AND NOT #AlwaysON;
END_REGION

REGION Network 3: CY52 interface L-UnloadingTransPalletLocationCylinder
   RUNG wire#powerrail
      Contact( #AlwaysON )
      wire#w1
      Contact( #E_stop )
      wire#w2
      Coil( "ST10Cylinder".Cy[52].In.GoWorkInterlock )
   END_RUNG
   RUNG wire#w2
      Coil( "ST10Cylinder".Cy[52].In.GoHomeInterlock )
   END_RUNG
   RUNG wire#w1
      I_Contact( #AlwaysON )
      Coil( "ST10Cylinder".Cy[52].In.Error )
   END_RUNG
   // the same network as SCL:
   "ST10Cylinder".Cy[52].In.GoWorkInterlock := #AlwaysON AND #E_stop;
   "ST10Cylinder".Cy[52].In.GoHomeInterlock := #AlwaysON AND #E_stop;
   "ST10Cylinder".Cy[52].In.Error := #AlwaysON AND NOT #AlwaysON;
END_REGION

REGION Network 4: CY53 interface L-UnloadingStopperCylinder1
   RUNG wire#powerrail
      Contact( #AlwaysON )
      wire#w1
      Contact( #E_stop )
      wire#w2
      Coil( "ST10Cylinder".Cy[53].In.GoWorkInterlock )
   END_RUNG
   RUNG wire#w2
      Coil( "ST10Cylinder".Cy[53].In.GoHomeInterlock )
   END_RUNG
   RUNG wire#w1
      I_Contact( #AlwaysON )
      Coil( "ST10Cylinder".Cy[53].In.Error )
   END_RUNG
   // the same network as SCL:
   "ST10Cylinder".Cy[53].In.GoWorkInterlock := #AlwaysON AND #E_stop;
   "ST10Cylinder".Cy[53].In.GoHomeInterlock := #AlwaysON AND #E_stop;
   "ST10Cylinder".Cy[53].In.Error := #AlwaysON AND NOT #AlwaysON;
END_REGION

REGION Network 5: CY54 interface L-UnloadingStopperCylinder2
   RUNG wire#powerrail
      Contact( #AlwaysON )
      wire#w1
      Contact( #E_stop )
      wire#w2
      Coil( "ST10Cylinder".Cy[54].In.GoWorkInterlock )
   END_RUNG
   RUNG wire#w2
      Coil( "ST10Cylinder".Cy[54].In.GoHomeInterlock )
   END_RUNG
   RUNG wire#w1
      I_Contact( #AlwaysON )
      Coil( "ST10Cylinder".Cy[54].In.Error )
   END_RUNG
   // the same network as SCL:
   "ST10Cylinder".Cy[54].In.GoWorkInterlock := #AlwaysON AND #E_stop;
   "ST10Cylinder".Cy[54].In.GoHomeInterlock := #AlwaysON AND #E_stop;
   "ST10Cylinder".Cy[54].In.Error := #AlwaysON AND NOT #AlwaysON;
END_REGION

REGION Network 6: CY55 interface L-UnloadingStopperCylinder3
   RUNG wire#powerrail
      Contact( #AlwaysON )
      wire#w1
      Contact( #E_stop )
      wire#w2
      Coil( "ST10Cylinder".Cy[55].In.GoWorkInterlock )
   END_RUNG
   RUNG wire#w2
      Coil( "ST10Cylinder".Cy[55].In.GoHomeInterlock )
   END_RUNG
   RUNG wire#w1
      I_Contact( #AlwaysON )
      Coil( "ST10Cylinder".Cy[55].In.Error )
   END_RUNG
   // the same network as SCL:
   "ST10Cylinder".Cy[55].In.GoWorkInterlock := #AlwaysON AND #E_stop;
   "ST10Cylinder".Cy[55].In.GoHomeInterlock := #AlwaysON AND #E_stop;
   "ST10Cylinder".Cy[55].In.Error := #AlwaysON AND NOT #AlwaysON;
END_REGION

REGION Network 7: CY56 interface
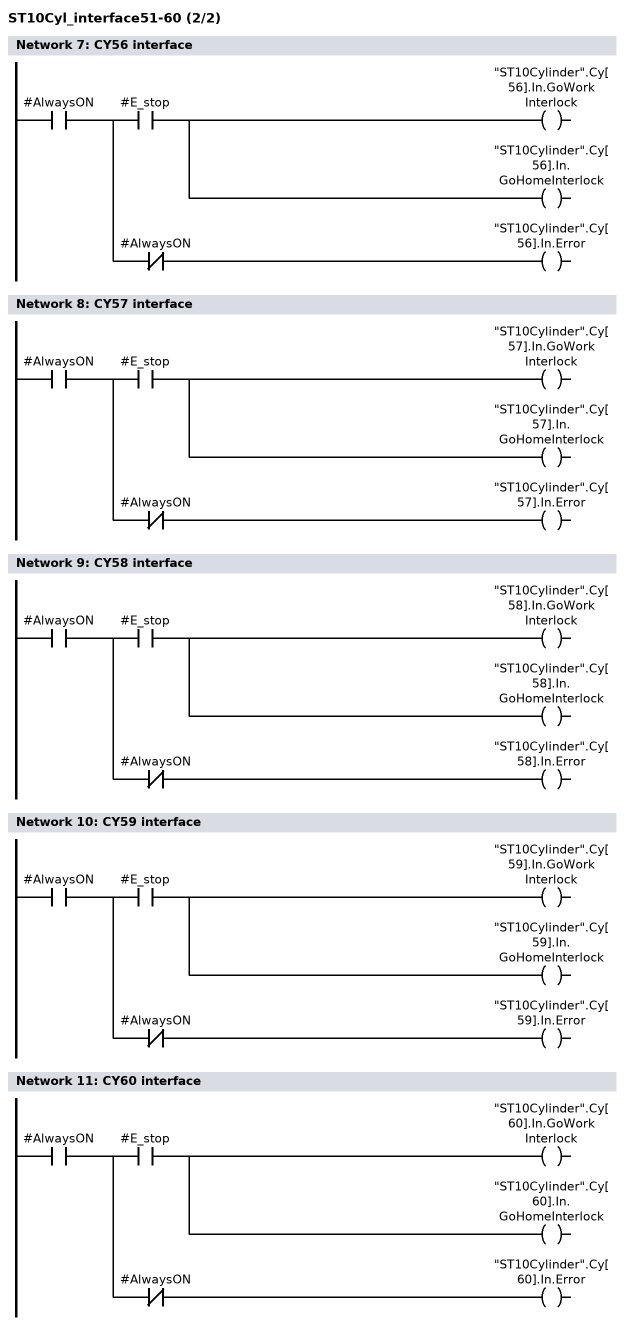
   RUNG wire#powerrail
      Contact( #AlwaysON )
      wire#w1
      Contact( #E_stop )
      wire#w2
      Coil( "ST10Cylinder".Cy[56].In.GoWorkInterlock )
   END_RUNG
   RUNG wire#w2
      Coil( "ST10Cylinder".Cy[56].In.GoHomeInterlock )
   END_RUNG
   RUNG wire#w1
      I_Contact( #AlwaysON )
      Coil( "ST10Cylinder".Cy[56].In.Error )
   END_RUNG
   // the same network as SCL:
   "ST10Cylinder".Cy[56].In.GoWorkInterlock := #AlwaysON AND #E_stop;
   "ST10Cylinder".Cy[56].In.GoHomeInterlock := #AlwaysON AND #E_stop;
   "ST10Cylinder".Cy[56].In.Error := #AlwaysON AND NOT #AlwaysON;
END_REGION

REGION Network 8: CY57 interface
   RUNG wire#powerrail
      Contact( #AlwaysON )
      wire#w1
      Contact( #E_stop )
      wire#w2
      Coil( "ST10Cylinder".Cy[57].In.GoWorkInterlock )
   END_RUNG
   RUNG wire#w2
      Coil( "ST10Cylinder".Cy[57].In.GoHomeInterlock )
   END_RUNG
   RUNG wire#w1
      I_Contact( #AlwaysON )
      Coil( "ST10Cylinder".Cy[57].In.Error )
   END_RUNG
   // the same network as SCL:
   "ST10Cylinder".Cy[57].In.GoWorkInterlock := #AlwaysON AND #E_stop;
   "ST10Cylinder".Cy[57].In.GoHomeInterlock := #AlwaysON AND #E_stop;
   "ST10Cylinder".Cy[57].In.Error := #AlwaysON AND NOT #AlwaysON;
END_REGION

REGION Network 9: CY58 interface
   RUNG wire#powerrail
      Contact( #AlwaysON )
      wire#w1
      Contact( #E_stop )
      wire#w2
      Coil( "ST10Cylinder".Cy[58].In.GoWorkInterlock )
   END_RUNG
   RUNG wire#w2
      Coil( "ST10Cylinder".Cy[58].In.GoHomeInterlock )
   END_RUNG
   RUNG wire#w1
      I_Contact( #AlwaysON )
      Coil( "ST10Cylinder".Cy[58].In.Error )
   END_RUNG
   // the same network as SCL:
   "ST10Cylinder".Cy[58].In.GoWorkInterlock := #AlwaysON AND #E_stop;
   "ST10Cylinder".Cy[58].In.GoHomeInterlock := #AlwaysON AND #E_stop;
   "ST10Cylinder".Cy[58].In.Error := #AlwaysON AND NOT #AlwaysON;
END_REGION

REGION Network 10: CY59 interface
   RUNG wire#powerrail
      Contact( #AlwaysON )
      wire#w1
      Contact( #E_stop )
      wire#w2
      Coil( "ST10Cylinder".Cy[59].In.GoWorkInterlock )
   END_RUNG
   RUNG wire#w2
      Coil( "ST10Cylinder".Cy[59].In.GoHomeInterlock )
   END_RUNG
   RUNG wire#w1
      I_Contact( #AlwaysON )
      Coil( "ST10Cylinder".Cy[59].In.Error )
   END_RUNG
   // the same network as SCL:
   "ST10Cylinder".Cy[59].In.GoWorkInterlock := #AlwaysON AND #E_stop;
   "ST10Cylinder".Cy[59].In.GoHomeInterlock := #AlwaysON AND #E_stop;
   "ST10Cylinder".Cy[59].In.Error := #AlwaysON AND NOT #AlwaysON;
END_REGION

REGION Network 11: CY60 interface
   RUNG wire#powerrail
      Contact( #AlwaysON )
      wire#w1
      Contact( #E_stop )
      wire#w2
      Coil( "ST10Cylinder".Cy[60].In.GoWorkInterlock )
   END_RUNG
   RUNG wire#w2
      Coil( "ST10Cylinder".Cy[60].In.GoHomeInterlock )
   END_RUNG
   RUNG wire#w1
      I_Contact( #AlwaysON )
      Coil( "ST10Cylinder".Cy[60].In.Error )
   END_RUNG
   // the same network as SCL:
   "ST10Cylinder".Cy[60].In.GoWorkInterlock := #AlwaysON AND #E_stop;
   "ST10Cylinder".Cy[60].In.GoHomeInterlock := #AlwaysON AND #E_stop;
   "ST10Cylinder".Cy[60].In.Error := #AlwaysON AND NOT #AlwaysON;
END_REGION
END_FUNCTION

FUNCTION "ST10Cyl_interface61-70" : Void   // FC1026, LAD
{ S7_Optimized_Access := 'FALSE' }
// stored: AutoNumber false, SetENOAutomatically false
   VAR_INPUT
      AlwaysON : Bool;
      E_stop : Bool;
   END_VAR
   VAR_TEMP
      tTest : Bool;
   END_VAR
BEGIN

REGION Network 1 (SCL): Cylinder 61-70 IO Interface (SCL)
   (*
   //Cylinder61 IO  K-reserveLifting3LiftingCylinder
   //Input
   "ST10Cylinder".Cy[61].In.WorkPositionSensor := "iK-reserveLifting3LiftingCylinderInWP";
   "ST10Cylinder".Cy[61].In.HomePositionSensor := "iK-reserveLifting3LiftingCylinderInHP";
   //Output
   "oK-reserveLifting3LiftingCylinderToWP" := "ST10Cylinder".Cy[61].Out.GoWorkPosition;
   "oK-reserveLifting3LiftingCylinderToHP" := "ST10Cylinder".Cy[61].Out.GoHomePosition;

   //Cylinder62 IO  K-reserveLifting3PalletLocationCylinder
   //Input
   "ST10Cylinder".Cy[62].In.WorkPositionSensor := "iK-reserveLifting3PalletLocationCylinderInWP";
   "ST10Cylinder".Cy[62].In.HomePositionSensor := "iK-reserveLifting3PalletLocationCylinderInHP";
   //Output
   "oK-reserveLifting3PalletLocationCylinderToWP" := "ST10Cylinder".Cy[62].Out.GoWorkPosition;
   "oK-reserveLifting3PalletLocationCylinderToHP" := "ST10Cylinder".Cy[62].Out.GoHomePosition;

   //Cylinder63 IO  K-reserveLoadingStopperCylinder1_1
   //Input
   "ST10Cylinder".Cy[63].In.WorkPositionSensor := "oK-reserveLoadingStopperCylinder1_1";
   "ST10Cylinder".Cy[63].In.HomePositionSensor := NOT "oK-reserveLoadingStopperCylinder1_1";
   //Output
   "oK-reserveLoadingStopperCylinder1_1" := "ST10Cylinder".Cy[63].Out.GoWorkPosition;
   //"oI-0030TrayLoading6trayStopperCylinderToHP" := "ST10Cylinder".Cy[63].Out.GoHomePosition;

   //Cylinder64 IO  K-reserveLoadingStopperCylinder1_2
   //Input
   "ST10Cylinder".Cy[64].In.WorkPositionSensor := "oK-reserveLoadingStopperCylinder1_2";
   "ST10Cylinder".Cy[64].In.HomePositionSensor := NOT "oK-reserveLoadingStopperCylinder1_2";
   //Output
   "oK-reserveLoadingStopperCylinder1_2" := "ST10Cylinder".Cy[64].Out.GoWorkPosition;
   //"oI-0060TrayLoadingTaketrayCylinderToHP" := "ST10Cylinder".Cy[64].Out.GoHomePosition;

   //Cylinder65 IO  K-reserveLoadingStopperCylinder2_1
   //Input
   "ST10Cylinder".Cy[65].In.WorkPositionSensor := "oK-reserveLoadingStopperCylinder2_1";
   "ST10Cylinder".Cy[65].In.HomePositionSensor := NOT "oK-reserveLoadingStopperCylinder2_1";
   //Output
   "oK-reserveLoadingStopperCylinder2_1" := "ST10Cylinder".Cy[65].Out.GoWorkPosition;
   //"oI-0050TrayLoadingTrayCylinderToHP" := "ST10Cylinder".Cy[65].Out.GoHomePosition;

   //Cylinder66 K-reserveLoadingStopperCylinder2_2
   //Input
   "ST10Cylinder".Cy[66].In.WorkPositionSensor := "oK-reserveLoadingStopperCylinder2_2";
   "ST10Cylinder".Cy[66].In.HomePositionSensor := NOT "oK-reserveLoadingStopperCylinder2_2";
   //Output
   "oK-reserveLoadingStopperCylinder2_2" := "ST10Cylinder".Cy[66].Out.GoWorkPosition;
   //"oI-0060TrayLoadingTraySupportCylinder1ToHP" := "ST10Cylinder".Cy[66].Out.GoHomePosition;

   //Cylinder67 K-reserveLoadingStopperCylinder3_1
   //Input
   "ST10Cylinder".Cy[67].In.WorkPositionSensor := "oK-reserveLoadingStopperCylinder3_1";
   "ST10Cylinder".Cy[67].In.HomePositionSensor := NOT "oK-reserveLoadingStopperCylinder3_1";
   //Output
   "oK-reserveLoadingStopperCylinder3_1" := "ST10Cylinder".Cy[67].Out.GoWorkPosition;
   //"oI-0070TrayLoadingTraySupportCylinder6ToHP" := "ST10Cylinder".Cy[67].Out.GoHomePosition;

   //Cylinder68 K-reserveLoadingStopperCylinder3_2
   //Input
   "ST10Cylinder".Cy[68].In.WorkPositionSensor := "oK-reserveLoadingStopperCylinder3_2";
   "ST10Cylinder".Cy[68].In.HomePositionSensor := NOT "oK-reserveLoadingStopperCylinder3_2";
   //Output
   "oK-reserveLoadingStopperCylinder3_2" := "ST10Cylinder".Cy[68].Out.GoWorkPosition;
   //"oI-0080TrayLoadingTrayLocationCylinderToHP" := "ST10Cylinder".Cy[68].Out.GoHomePosition;

   //Cylinder69 K-reserveLoadingStopperCylinder4_1
   //Input
   "ST10Cylinder".Cy[69].In.WorkPositionSensor := "oK-reserveLoadingStopperCylinder4_1";
   "ST10Cylinder".Cy[69].In.HomePositionSensor := NOT "oK-reserveLoadingStopperCylinder4_1";
   //Output
   "oK-reserveLoadingStopperCylinder4_1" := "ST10Cylinder".Cy[69].Out.GoWorkPosition;
   //"oI-0090TrayLoadingTrayUnloadingLiftingCylinderToHP" := "ST10Cylinder".Cy[69].Out.GoHomePosition;

   //Cylinder70 K-reserveLoadingStopperCylinder4_2
   // //Input
   "ST10Cylinder".Cy[70].In.WorkPositionSensor := "oK-reserveLoadingStopperCylinder4_2";
   "ST10Cylinder".Cy[70].In.HomePositionSensor := NOT "oK-reserveLoadingStopperCylinder4_2";
   // //Output
   "oK-reserveLoadingStopperCylinder4_2" := "ST10Cylinder".Cy[70].Out.GoWorkPosition;
   // "Feeding washer  lift Cylinder ToHP" := "ST10Cylinder".Cy[70].Out.GoHomePosition;
   *)
END_REGION

REGION Network 2: CY61 interface K-reserveLifting3LiftingCylinder
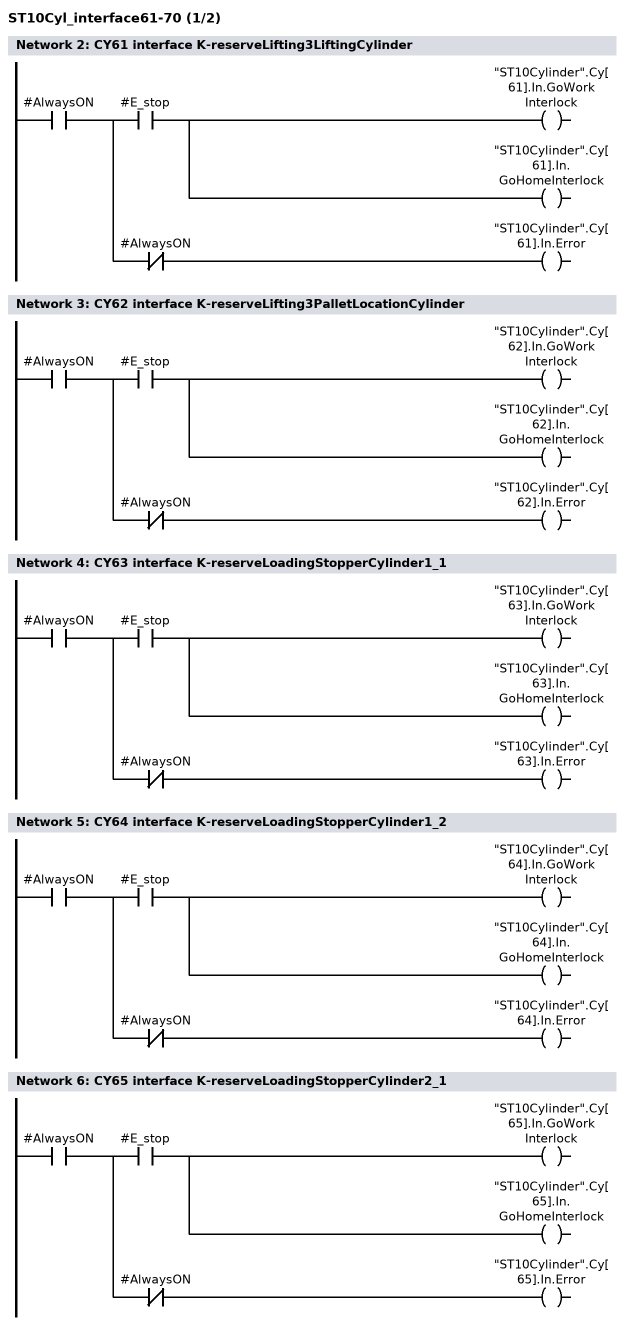
   RUNG wire#powerrail
      Contact( #AlwaysON )
      wire#w1
      Contact( #E_stop )
      wire#w2
      Coil( "ST10Cylinder".Cy[61].In.GoWorkInterlock )
   END_RUNG
   RUNG wire#w2
      Coil( "ST10Cylinder".Cy[61].In.GoHomeInterlock )
   END_RUNG
   RUNG wire#w1
      I_Contact( #AlwaysON )
      Coil( "ST10Cylinder".Cy[61].In.Error )
   END_RUNG
   // the same network as SCL:
   "ST10Cylinder".Cy[61].In.GoWorkInterlock := #AlwaysON AND #E_stop;
   "ST10Cylinder".Cy[61].In.GoHomeInterlock := #AlwaysON AND #E_stop;
   "ST10Cylinder".Cy[61].In.Error := #AlwaysON AND NOT #AlwaysON;
END_REGION

REGION Network 3: CY62 interface K-reserveLifting3PalletLocationCylinder
   RUNG wire#powerrail
      Contact( #AlwaysON )
      wire#w1
      Contact( #E_stop )
      wire#w2
      Coil( "ST10Cylinder".Cy[62].In.GoWorkInterlock )
   END_RUNG
   RUNG wire#w2
      Coil( "ST10Cylinder".Cy[62].In.GoHomeInterlock )
   END_RUNG
   RUNG wire#w1
      I_Contact( #AlwaysON )
      Coil( "ST10Cylinder".Cy[62].In.Error )
   END_RUNG
   // the same network as SCL:
   "ST10Cylinder".Cy[62].In.GoWorkInterlock := #AlwaysON AND #E_stop;
   "ST10Cylinder".Cy[62].In.GoHomeInterlock := #AlwaysON AND #E_stop;
   "ST10Cylinder".Cy[62].In.Error := #AlwaysON AND NOT #AlwaysON;
END_REGION

REGION Network 4: CY63 interface K-reserveLoadingStopperCylinder1_1
   RUNG wire#powerrail
      Contact( #AlwaysON )
      wire#w1
      Contact( #E_stop )
      wire#w2
      Coil( "ST10Cylinder".Cy[63].In.GoWorkInterlock )
   END_RUNG
   RUNG wire#w2
      Coil( "ST10Cylinder".Cy[63].In.GoHomeInterlock )
   END_RUNG
   RUNG wire#w1
      I_Contact( #AlwaysON )
      Coil( "ST10Cylinder".Cy[63].In.Error )
   END_RUNG
   // the same network as SCL:
   "ST10Cylinder".Cy[63].In.GoWorkInterlock := #AlwaysON AND #E_stop;
   "ST10Cylinder".Cy[63].In.GoHomeInterlock := #AlwaysON AND #E_stop;
   "ST10Cylinder".Cy[63].In.Error := #AlwaysON AND NOT #AlwaysON;
END_REGION

REGION Network 5: CY64 interface K-reserveLoadingStopperCylinder1_2
   RUNG wire#powerrail
      Contact( #AlwaysON )
      wire#w1
      Contact( #E_stop )
      wire#w2
      Coil( "ST10Cylinder".Cy[64].In.GoWorkInterlock )
   END_RUNG
   RUNG wire#w2
      Coil( "ST10Cylinder".Cy[64].In.GoHomeInterlock )
   END_RUNG
   RUNG wire#w1
      I_Contact( #AlwaysON )
      Coil( "ST10Cylinder".Cy[64].In.Error )
   END_RUNG
   // the same network as SCL:
   "ST10Cylinder".Cy[64].In.GoWorkInterlock := #AlwaysON AND #E_stop;
   "ST10Cylinder".Cy[64].In.GoHomeInterlock := #AlwaysON AND #E_stop;
   "ST10Cylinder".Cy[64].In.Error := #AlwaysON AND NOT #AlwaysON;
END_REGION

REGION Network 6: CY65 interface K-reserveLoadingStopperCylinder2_1
   RUNG wire#powerrail
      Contact( #AlwaysON )
      wire#w1
      Contact( #E_stop )
      wire#w2
      Coil( "ST10Cylinder".Cy[65].In.GoWorkInterlock )
   END_RUNG
   RUNG wire#w2
      Coil( "ST10Cylinder".Cy[65].In.GoHomeInterlock )
   END_RUNG
   RUNG wire#w1
      I_Contact( #AlwaysON )
      Coil( "ST10Cylinder".Cy[65].In.Error )
   END_RUNG
   // the same network as SCL:
   "ST10Cylinder".Cy[65].In.GoWorkInterlock := #AlwaysON AND #E_stop;
   "ST10Cylinder".Cy[65].In.GoHomeInterlock := #AlwaysON AND #E_stop;
   "ST10Cylinder".Cy[65].In.Error := #AlwaysON AND NOT #AlwaysON;
END_REGION

REGION Network 7: CY66 interface K-reserveLoadingStopperCylinder2_2
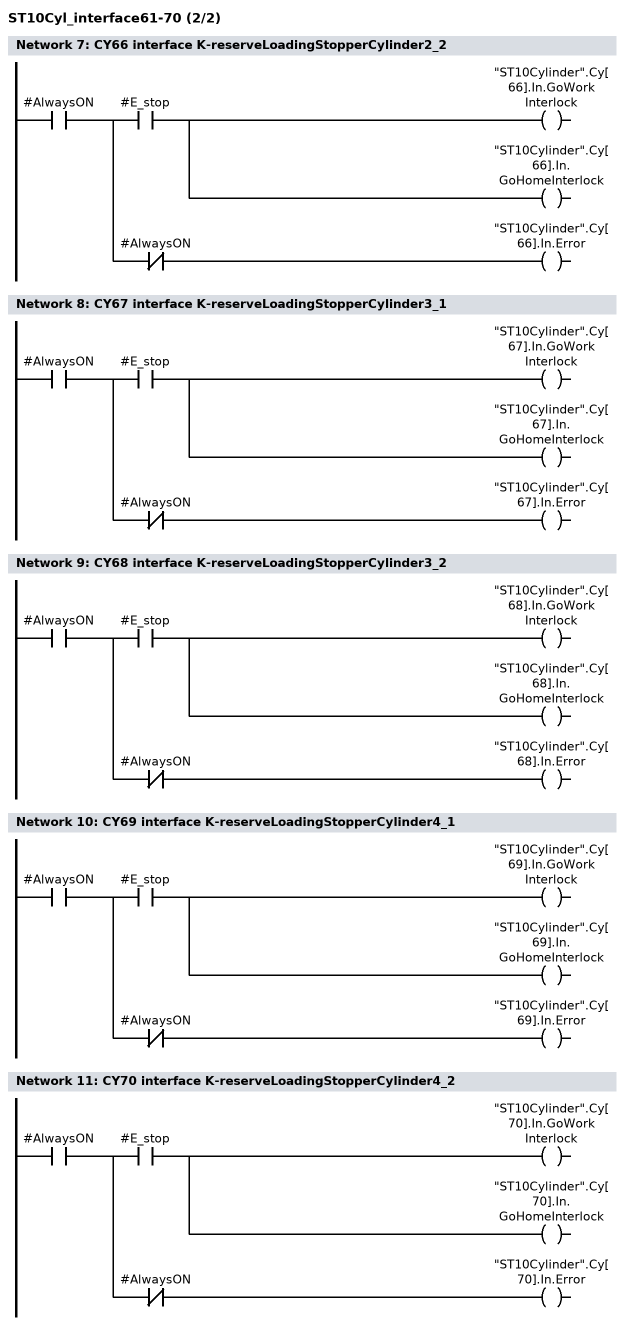
   RUNG wire#powerrail
      Contact( #AlwaysON )
      wire#w1
      Contact( #E_stop )
      wire#w2
      Coil( "ST10Cylinder".Cy[66].In.GoWorkInterlock )
   END_RUNG
   RUNG wire#w2
      Coil( "ST10Cylinder".Cy[66].In.GoHomeInterlock )
   END_RUNG
   RUNG wire#w1
      I_Contact( #AlwaysON )
      Coil( "ST10Cylinder".Cy[66].In.Error )
   END_RUNG
   // the same network as SCL:
   "ST10Cylinder".Cy[66].In.GoWorkInterlock := #AlwaysON AND #E_stop;
   "ST10Cylinder".Cy[66].In.GoHomeInterlock := #AlwaysON AND #E_stop;
   "ST10Cylinder".Cy[66].In.Error := #AlwaysON AND NOT #AlwaysON;
END_REGION

REGION Network 8: CY67 interface K-reserveLoadingStopperCylinder3_1
   RUNG wire#powerrail
      Contact( #AlwaysON )
      wire#w1
      Contact( #E_stop )
      wire#w2
      Coil( "ST10Cylinder".Cy[67].In.GoWorkInterlock )
   END_RUNG
   RUNG wire#w2
      Coil( "ST10Cylinder".Cy[67].In.GoHomeInterlock )
   END_RUNG
   RUNG wire#w1
      I_Contact( #AlwaysON )
      Coil( "ST10Cylinder".Cy[67].In.Error )
   END_RUNG
   // the same network as SCL:
   "ST10Cylinder".Cy[67].In.GoWorkInterlock := #AlwaysON AND #E_stop;
   "ST10Cylinder".Cy[67].In.GoHomeInterlock := #AlwaysON AND #E_stop;
   "ST10Cylinder".Cy[67].In.Error := #AlwaysON AND NOT #AlwaysON;
END_REGION

REGION Network 9: CY68 interface K-reserveLoadingStopperCylinder3_2
   RUNG wire#powerrail
      Contact( #AlwaysON )
      wire#w1
      Contact( #E_stop )
      wire#w2
      Coil( "ST10Cylinder".Cy[68].In.GoWorkInterlock )
   END_RUNG
   RUNG wire#w2
      Coil( "ST10Cylinder".Cy[68].In.GoHomeInterlock )
   END_RUNG
   RUNG wire#w1
      I_Contact( #AlwaysON )
      Coil( "ST10Cylinder".Cy[68].In.Error )
   END_RUNG
   // the same network as SCL:
   "ST10Cylinder".Cy[68].In.GoWorkInterlock := #AlwaysON AND #E_stop;
   "ST10Cylinder".Cy[68].In.GoHomeInterlock := #AlwaysON AND #E_stop;
   "ST10Cylinder".Cy[68].In.Error := #AlwaysON AND NOT #AlwaysON;
END_REGION

REGION Network 10: CY69 interface K-reserveLoadingStopperCylinder4_1
   RUNG wire#powerrail
      Contact( #AlwaysON )
      wire#w1
      Contact( #E_stop )
      wire#w2
      Coil( "ST10Cylinder".Cy[69].In.GoWorkInterlock )
   END_RUNG
   RUNG wire#w2
      Coil( "ST10Cylinder".Cy[69].In.GoHomeInterlock )
   END_RUNG
   RUNG wire#w1
      I_Contact( #AlwaysON )
      Coil( "ST10Cylinder".Cy[69].In.Error )
   END_RUNG
   // the same network as SCL:
   "ST10Cylinder".Cy[69].In.GoWorkInterlock := #AlwaysON AND #E_stop;
   "ST10Cylinder".Cy[69].In.GoHomeInterlock := #AlwaysON AND #E_stop;
   "ST10Cylinder".Cy[69].In.Error := #AlwaysON AND NOT #AlwaysON;
END_REGION

REGION Network 11: CY70 interface K-reserveLoadingStopperCylinder4_2
   RUNG wire#powerrail
      Contact( #AlwaysON )
      wire#w1
      Contact( #E_stop )
      wire#w2
      Coil( "ST10Cylinder".Cy[70].In.GoWorkInterlock )
   END_RUNG
   RUNG wire#w2
      Coil( "ST10Cylinder".Cy[70].In.GoHomeInterlock )
   END_RUNG
   RUNG wire#w1
      I_Contact( #AlwaysON )
      Coil( "ST10Cylinder".Cy[70].In.Error )
   END_RUNG
   // the same network as SCL:
   "ST10Cylinder".Cy[70].In.GoWorkInterlock := #AlwaysON AND #E_stop;
   "ST10Cylinder".Cy[70].In.GoHomeInterlock := #AlwaysON AND #E_stop;
   "ST10Cylinder".Cy[70].In.Error := #AlwaysON AND NOT #AlwaysON;
END_REGION
END_FUNCTION

FUNCTION "ST10Cyl_interface71-80" : Void   // FC1027, LAD
{ S7_Optimized_Access := 'FALSE' }
// stored: AutoNumber false, SetENOAutomatically false
   VAR_INPUT
      AlwaysON : Bool;
      E_stop : Bool;
   END_VAR
   VAR_TEMP
      tTest : Bool;
   END_VAR
BEGIN

REGION Network 1 (SCL): Cylinder 71-80 IO Interface (SCL)
   (*
   //Cylinder71 IO    K-reserveTakeStopperCylinder1_1
   //Input
   "ST10Cylinder".Cy[71].In.WorkPositionSensor := "oK-reserveTakeStopperCylinder1_1";
   "ST10Cylinder".Cy[71].In.HomePositionSensor := NOT "oK-reserveTakeStopperCylinder1_1";
   //Output
   "oK-reserveTakeStopperCylinder1_1" := "ST10Cylinder".Cy[71].Out.GoWorkPosition;
   #tTest := "ST10Cylinder".Cy[71].Out.GoHomePosition;

   //Cylinder72 IO    K-reserveTakeStopperCylinder1_2
   //Input
   "ST10Cylinder".Cy[72].In.WorkPositionSensor := "oK-reserveTakeStopperCylinder1_2";
   "ST10Cylinder".Cy[72].In.HomePositionSensor := NOT "oK-reserveTakeStopperCylinder1_2";
   //Output
   "oK-reserveTakeStopperCylinder1_2" := "ST10Cylinder".Cy[72].Out.GoWorkPosition;
   #tTest := "ST10Cylinder".Cy[72].Out.GoHomePosition;

   //Cylinder73 IO  K-reserveTakeStopperCylinder2_1
   //Input
   "ST10Cylinder".Cy[73].In.WorkPositionSensor := "oK-reserveTakeStopperCylinder2_1";
   "ST10Cylinder".Cy[73].In.HomePositionSensor := NOT "oK-reserveTakeStopperCylinder2_1";
   //Output
   "oK-reserveTakeStopperCylinder2_1" := "ST10Cylinder".Cy[73].Out.GoWorkPosition;
   #tTest := "ST10Cylinder".Cy[73].Out.GoHomePosition;

   //Cylinder74 IO  K-reserveTakeStopperCylinder2_2
   //Input
   "ST10Cylinder".Cy[74].In.WorkPositionSensor := "oK-reserveTakeStopperCylinder2_2";
   "ST10Cylinder".Cy[74].In.HomePositionSensor := NOT "oK-reserveTakeStopperCylinder2_2";
   //Output
   "oK-reserveTakeStopperCylinder2_2" := "ST10Cylinder".Cy[74].Out.GoWorkPosition;
   #tTest := "ST10Cylinder".Cy[74].Out.GoHomePosition;

   //Cylinder75 IO  K-reserveTakeStopperCylinder3_1
   //Input
   "ST10Cylinder".Cy[75].In.WorkPositionSensor := "oK-reserveTakeStopperCylinder3_1";
   "ST10Cylinder".Cy[75].In.HomePositionSensor := NOT "oK-reserveTakeStopperCylinder3_1";
   //Output
   "oK-reserveTakeStopperCylinder3_1" := "ST10Cylinder".Cy[75].Out.GoWorkPosition;
   #tTest := "ST10Cylinder".Cy[75].Out.GoHomePosition;

   //Cylinder76 IO  K-reserveTakeStopperCylinder3_2
   //Input
   "ST10Cylinder".Cy[76].In.WorkPositionSensor := "oK-reserveTakeStopperCylinder3_2";
   "ST10Cylinder".Cy[76].In.HomePositionSensor := NOT "oK-reserveTakeStopperCylinder3_2";
   //Output
   "oK-reserveTakeStopperCylinder3_2" := "ST10Cylinder".Cy[76].Out.GoWorkPosition;
   #tTest := "ST10Cylinder".Cy[76].Out.GoHomePosition;

   *)
END_REGION

REGION Network 2: CY71 interface K-reserveTakeStopperCylinder1_1
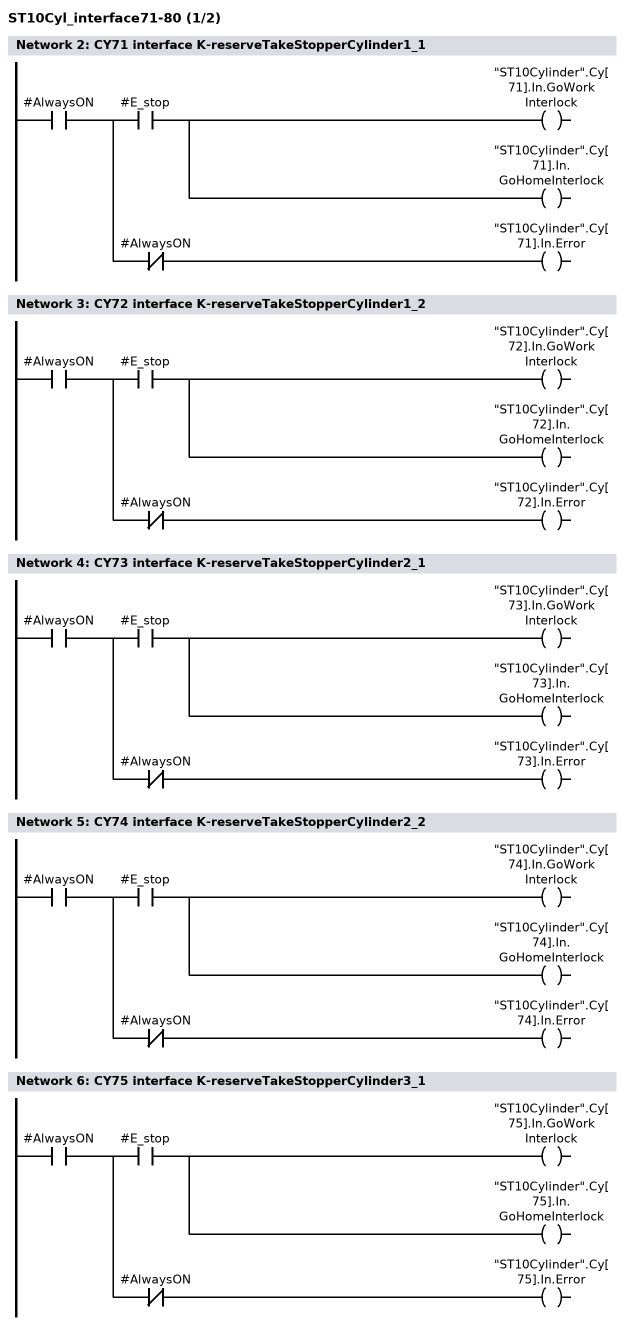
   RUNG wire#powerrail
      Contact( #AlwaysON )
      wire#w1
      Contact( #E_stop )
      wire#w2
      Coil( "ST10Cylinder".Cy[71].In.GoWorkInterlock )
   END_RUNG
   RUNG wire#w2
      Coil( "ST10Cylinder".Cy[71].In.GoHomeInterlock )
   END_RUNG
   RUNG wire#w1
      I_Contact( #AlwaysON )
      Coil( "ST10Cylinder".Cy[71].In.Error )
   END_RUNG
   // the same network as SCL:
   "ST10Cylinder".Cy[71].In.GoWorkInterlock := #AlwaysON AND #E_stop;
   "ST10Cylinder".Cy[71].In.GoHomeInterlock := #AlwaysON AND #E_stop;
   "ST10Cylinder".Cy[71].In.Error := #AlwaysON AND NOT #AlwaysON;
END_REGION

REGION Network 3: CY72 interface K-reserveTakeStopperCylinder1_2
   RUNG wire#powerrail
      Contact( #AlwaysON )
      wire#w1
      Contact( #E_stop )
      wire#w2
      Coil( "ST10Cylinder".Cy[72].In.GoWorkInterlock )
   END_RUNG
   RUNG wire#w2
      Coil( "ST10Cylinder".Cy[72].In.GoHomeInterlock )
   END_RUNG
   RUNG wire#w1
      I_Contact( #AlwaysON )
      Coil( "ST10Cylinder".Cy[72].In.Error )
   END_RUNG
   // the same network as SCL:
   "ST10Cylinder".Cy[72].In.GoWorkInterlock := #AlwaysON AND #E_stop;
   "ST10Cylinder".Cy[72].In.GoHomeInterlock := #AlwaysON AND #E_stop;
   "ST10Cylinder".Cy[72].In.Error := #AlwaysON AND NOT #AlwaysON;
END_REGION

REGION Network 4: CY73 interface K-reserveTakeStopperCylinder2_1
   RUNG wire#powerrail
      Contact( #AlwaysON )
      wire#w1
      Contact( #E_stop )
      wire#w2
      Coil( "ST10Cylinder".Cy[73].In.GoWorkInterlock )
   END_RUNG
   RUNG wire#w2
      Coil( "ST10Cylinder".Cy[73].In.GoHomeInterlock )
   END_RUNG
   RUNG wire#w1
      I_Contact( #AlwaysON )
      Coil( "ST10Cylinder".Cy[73].In.Error )
   END_RUNG
   // the same network as SCL:
   "ST10Cylinder".Cy[73].In.GoWorkInterlock := #AlwaysON AND #E_stop;
   "ST10Cylinder".Cy[73].In.GoHomeInterlock := #AlwaysON AND #E_stop;
   "ST10Cylinder".Cy[73].In.Error := #AlwaysON AND NOT #AlwaysON;
END_REGION

REGION Network 5: CY74 interface K-reserveTakeStopperCylinder2_2
   RUNG wire#powerrail
      Contact( #AlwaysON )
      wire#w1
      Contact( #E_stop )
      wire#w2
      Coil( "ST10Cylinder".Cy[74].In.GoWorkInterlock )
   END_RUNG
   RUNG wire#w2
      Coil( "ST10Cylinder".Cy[74].In.GoHomeInterlock )
   END_RUNG
   RUNG wire#w1
      I_Contact( #AlwaysON )
      Coil( "ST10Cylinder".Cy[74].In.Error )
   END_RUNG
   // the same network as SCL:
   "ST10Cylinder".Cy[74].In.GoWorkInterlock := #AlwaysON AND #E_stop;
   "ST10Cylinder".Cy[74].In.GoHomeInterlock := #AlwaysON AND #E_stop;
   "ST10Cylinder".Cy[74].In.Error := #AlwaysON AND NOT #AlwaysON;
END_REGION

REGION Network 6: CY75 interface K-reserveTakeStopperCylinder3_1
   RUNG wire#powerrail
      Contact( #AlwaysON )
      wire#w1
      Contact( #E_stop )
      wire#w2
      Coil( "ST10Cylinder".Cy[75].In.GoWorkInterlock )
   END_RUNG
   RUNG wire#w2
      Coil( "ST10Cylinder".Cy[75].In.GoHomeInterlock )
   END_RUNG
   RUNG wire#w1
      I_Contact( #AlwaysON )
      Coil( "ST10Cylinder".Cy[75].In.Error )
   END_RUNG
   // the same network as SCL:
   "ST10Cylinder".Cy[75].In.GoWorkInterlock := #AlwaysON AND #E_stop;
   "ST10Cylinder".Cy[75].In.GoHomeInterlock := #AlwaysON AND #E_stop;
   "ST10Cylinder".Cy[75].In.Error := #AlwaysON AND NOT #AlwaysON;
END_REGION

REGION Network 7: CY76 interface K-reserveTakeStopperCylinder3_2
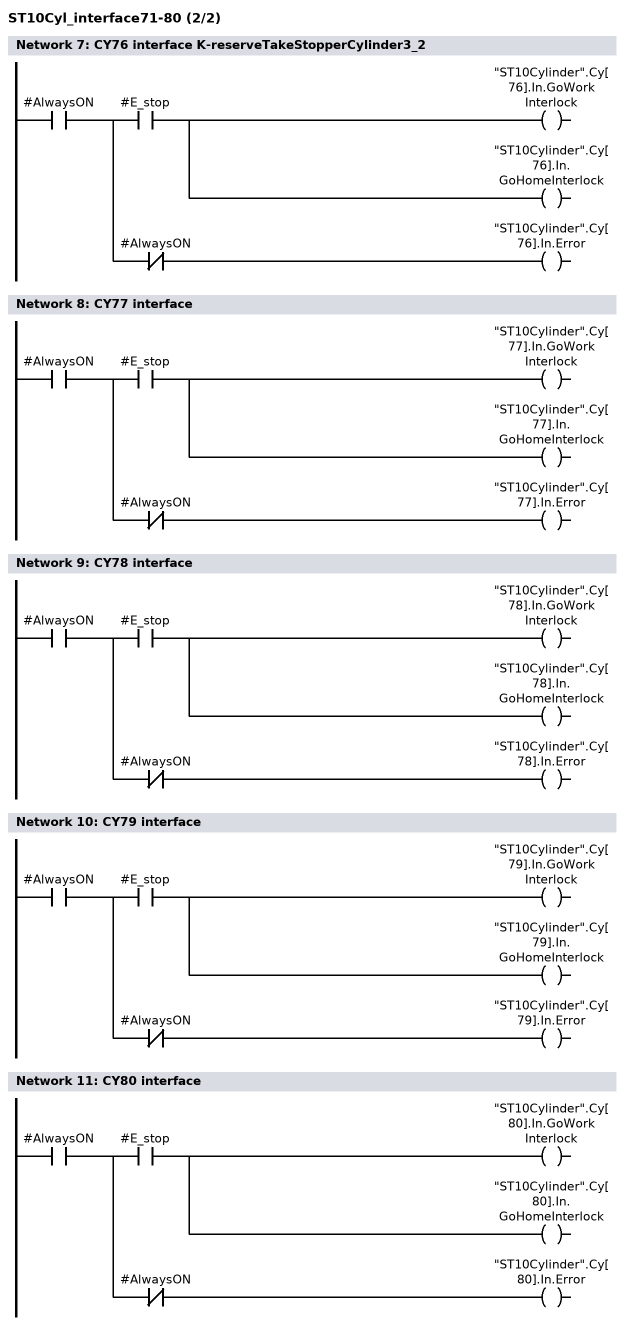
   RUNG wire#powerrail
      Contact( #AlwaysON )
      wire#w1
      Contact( #E_stop )
      wire#w2
      Coil( "ST10Cylinder".Cy[76].In.GoWorkInterlock )
   END_RUNG
   RUNG wire#w2
      Coil( "ST10Cylinder".Cy[76].In.GoHomeInterlock )
   END_RUNG
   RUNG wire#w1
      I_Contact( #AlwaysON )
      Coil( "ST10Cylinder".Cy[76].In.Error )
   END_RUNG
   // the same network as SCL:
   "ST10Cylinder".Cy[76].In.GoWorkInterlock := #AlwaysON AND #E_stop;
   "ST10Cylinder".Cy[76].In.GoHomeInterlock := #AlwaysON AND #E_stop;
   "ST10Cylinder".Cy[76].In.Error := #AlwaysON AND NOT #AlwaysON;
END_REGION

REGION Network 8: CY77 interface
   RUNG wire#powerrail
      Contact( #AlwaysON )
      wire#w1
      Contact( #E_stop )
      wire#w2
      Coil( "ST10Cylinder".Cy[77].In.GoWorkInterlock )
   END_RUNG
   RUNG wire#w2
      Coil( "ST10Cylinder".Cy[77].In.GoHomeInterlock )
   END_RUNG
   RUNG wire#w1
      I_Contact( #AlwaysON )
      Coil( "ST10Cylinder".Cy[77].In.Error )
   END_RUNG
   // the same network as SCL:
   "ST10Cylinder".Cy[77].In.GoWorkInterlock := #AlwaysON AND #E_stop;
   "ST10Cylinder".Cy[77].In.GoHomeInterlock := #AlwaysON AND #E_stop;
   "ST10Cylinder".Cy[77].In.Error := #AlwaysON AND NOT #AlwaysON;
END_REGION

REGION Network 9: CY78 interface
   RUNG wire#powerrail
      Contact( #AlwaysON )
      wire#w1
      Contact( #E_stop )
      wire#w2
      Coil( "ST10Cylinder".Cy[78].In.GoWorkInterlock )
   END_RUNG
   RUNG wire#w2
      Coil( "ST10Cylinder".Cy[78].In.GoHomeInterlock )
   END_RUNG
   RUNG wire#w1
      I_Contact( #AlwaysON )
      Coil( "ST10Cylinder".Cy[78].In.Error )
   END_RUNG
   // the same network as SCL:
   "ST10Cylinder".Cy[78].In.GoWorkInterlock := #AlwaysON AND #E_stop;
   "ST10Cylinder".Cy[78].In.GoHomeInterlock := #AlwaysON AND #E_stop;
   "ST10Cylinder".Cy[78].In.Error := #AlwaysON AND NOT #AlwaysON;
END_REGION

REGION Network 10: CY79 interface
   RUNG wire#powerrail
      Contact( #AlwaysON )
      wire#w1
      Contact( #E_stop )
      wire#w2
      Coil( "ST10Cylinder".Cy[79].In.GoWorkInterlock )
   END_RUNG
   RUNG wire#w2
      Coil( "ST10Cylinder".Cy[79].In.GoHomeInterlock )
   END_RUNG
   RUNG wire#w1
      I_Contact( #AlwaysON )
      Coil( "ST10Cylinder".Cy[79].In.Error )
   END_RUNG
   // the same network as SCL:
   "ST10Cylinder".Cy[79].In.GoWorkInterlock := #AlwaysON AND #E_stop;
   "ST10Cylinder".Cy[79].In.GoHomeInterlock := #AlwaysON AND #E_stop;
   "ST10Cylinder".Cy[79].In.Error := #AlwaysON AND NOT #AlwaysON;
END_REGION

REGION Network 11: CY80 interface
   RUNG wire#powerrail
      Contact( #AlwaysON )
      wire#w1
      Contact( #E_stop )
      wire#w2
      Coil( "ST10Cylinder".Cy[80].In.GoWorkInterlock )
   END_RUNG
   RUNG wire#w2
      Coil( "ST10Cylinder".Cy[80].In.GoHomeInterlock )
   END_RUNG
   RUNG wire#w1
      I_Contact( #AlwaysON )
      Coil( "ST10Cylinder".Cy[80].In.Error )
   END_RUNG
   // the same network as SCL:
   "ST10Cylinder".Cy[80].In.GoWorkInterlock := #AlwaysON AND #E_stop;
   "ST10Cylinder".Cy[80].In.GoHomeInterlock := #AlwaysON AND #E_stop;
   "ST10Cylinder".Cy[80].In.Error := #AlwaysON AND NOT #AlwaysON;
END_REGION
END_FUNCTION

FUNCTION "ST10Cyl_interface81-90" : Void   // FC1028, LAD
{ S7_Optimized_Access := 'FALSE' }
VERSION : 0.1
// stored: AutoNumber false, IsIECCheckEnabled false, SetENOAutomatically false, UDAEnableTagReadback false
   VAR_INPUT
      AlwaysON : Bool;
      E_stop : Bool;
   END_VAR
   VAR_TEMP
      tTest : Bool;
   END_VAR
BEGIN

REGION Network 1 (SCL): Cylinder 81-90 IO Interface (SCL)
   (*
   //Cylinder81 IO  L-UnloadingTransCylinder
   //Input
   "ST10Cylinder".Cy[81].In.WorkPositionSensor := "iL-UnloadingTransCylinderInWP";
   "ST10Cylinder".Cy[81].In.HomePositionSensor := "iL-UnloadingTransCylinderInHP";
   //Output
   "oL-UnloadingTransCylinderToWP" := "ST10Cylinder".Cy[81].Out.GoWorkPosition;
   "oL-UnloadingTransCylinderToHP" := "ST10Cylinder".Cy[81].Out.GoHomePosition;

   //Cylinder82 IO  L-UnloadingTransPalletLocationCylinder
   //Input
   "ST10Cylinder".Cy[82].In.WorkPositionSensor := "iL-UnloadingTransPalletLocationCylinderInWP";
   "ST10Cylinder".Cy[82].In.HomePositionSensor := "iL-UnloadingTransPalletLocationCylinderInHP";
   //Output
   "oL-UnloadingTransPalletLocationCylinderToWP" := "ST10Cylinder".Cy[82].Out.GoWorkPosition;
   "oL-UnloadingTransPalletLocationCylinderToHP" := "ST10Cylinder".Cy[82].Out.GoHomePosition;

   //Cylinder83 IO  L-UnloadingStopperCylinder1_1
   //Input
   "ST10Cylinder".Cy[83].In.WorkPositionSensor := "oL-UnloadingStopperCylinder1_1";
   "ST10Cylinder".Cy[83].In.HomePositionSensor := NOT "oL-UnloadingStopperCylinder1_1";
   //Output
   "oL-UnloadingStopperCylinder1_1" := "ST10Cylinder".Cy[83].Out.GoWorkPosition;
   //"oI-0030TrayLoading8trayStopperCylinderToHP" := "ST10Cylinder".Cy[83].Out.GoHomePosition;

   //Cylinder84 IO  L-UnloadingStopperCylinder1_2
   //Input
   "ST10Cylinder".Cy[84].In.WorkPositionSensor := "oL-UnloadingStopperCylinder1_2";
   "ST10Cylinder".Cy[84].In.HomePositionSensor := NOT "oL-UnloadingStopperCylinder1_2";
   //Output
   "oL-UnloadingStopperCylinder1_2" := "ST10Cylinder".Cy[84].Out.GoWorkPosition;
   //"oI-0080TrayLoadingTaketrayCylinderToHP" := "ST10Cylinder".Cy[84].Out.GoHomePosition;

   //Cylinder85 IO  L-UnloadingStopperCylinder2_1
   //Input
   "ST10Cylinder".Cy[85].In.WorkPositionSensor := "oL-UnloadingStopperCylinder2_1";
   "ST10Cylinder".Cy[85].In.HomePositionSensor := NOT "oL-UnloadingStopperCylinder2_1";
   //Output
   "oL-UnloadingStopperCylinder2_1" := "ST10Cylinder".Cy[85].Out.GoWorkPosition;
   //"oI-0050TrayLoadingTrayCylinderToHP" := "ST10Cylinder".Cy[85].Out.GoHomePosition;

   //Cylinder86  L-UnloadingStopperCylinder2_2
   //Input
   "ST10Cylinder".Cy[86].In.WorkPositionSensor := "oL-UnloadingStopperCylinder2_2";
   "ST10Cylinder".Cy[86].In.HomePositionSensor := NOT "oL-UnloadingStopperCylinder2_2";
   //Output
   "oL-UnloadingStopperCylinder2_2" := "ST10Cylinder".Cy[86].Out.GoWorkPosition;
   //"oI-0080TrayLoadingTraySupportCylinder1ToHP" := "ST10Cylinder".Cy[86].Out.GoHomePosition;

   //Cylinder87 L-UnloadingStopperCylinder3_1
   //Input
   "ST10Cylinder".Cy[87].In.WorkPositionSensor := "oL-UnloadingStopperCylinder3_1";
   "ST10Cylinder".Cy[87].In.HomePositionSensor := NOT "oL-UnloadingStopperCylinder3_1";
   //Output
   "oL-UnloadingStopperCylinder3_1" := "ST10Cylinder".Cy[87].Out.GoWorkPosition;
   //"oI-0070TrayLoadingTraySupportCylinder8ToHP" := "ST10Cylinder".Cy[87].Out.GoHomePosition;

   //Cylinder88 L-UnloadingStopperCylinder3_2
   //Input
   "ST10Cylinder".Cy[88].In.WorkPositionSensor := "oL-UnloadingStopperCylinder3_2";
   "ST10Cylinder".Cy[88].In.HomePositionSensor := NOT "oL-UnloadingStopperCylinder3_2";
   //Output
   "oL-UnloadingStopperCylinder3_2" := "ST10Cylinder".Cy[88].Out.GoWorkPosition;
   //"oI-0080TrayLoadingTrayLocationCylinderToHP" := "ST10Cylinder".Cy[88].Out.GoHomePosition;
   //
   *)
   (*
   //Cylinder89 K-reserveLoadingStopperCylinder4_1
   //Input
   "ST10Cylinder".Cy[89].In.WorkPositionSensor := "oK-reserveLoadingStopperCylinder4_1";
   "ST10Cylinder".Cy[89].In.HomePositionSensor := NOT "oK-reserveLoadingStopperCylinder4_1";
   //Output
   "oK-reserveLoadingStopperCylinder4_1" := "ST10Cylinder".Cy[89].Out.GoWorkPosition;
   //"oI-0090TrayLoadingTrayUnloadingLiftingCylinderToHP" := "ST10Cylinder".Cy[89].Out.GoHomePosition;

   //Cylinder70 K-reserveLoadingStopperCylinder4_2
   // //Input
   "ST10Cylinder".Cy[70].In.WorkPositionSensor := "oK-reserveLoadingStopperCylinder4_2";
   "ST10Cylinder".Cy[70].In.HomePositionSensor := NOT "oK-reserveLoadingStopperCylinder4_2";
   // //Output
   "oK-reserveLoadingStopperCylinder4_2" := "ST10Cylinder".Cy[70].Out.GoWorkPosition;
   // "Feeding washer  lift Cylinder ToHP" := "ST10Cylinder".Cy[70].Out.GoHomePosition;

   *)
END_REGION

REGION Network 2: CY81 interface L-UnloadingTransCylinder
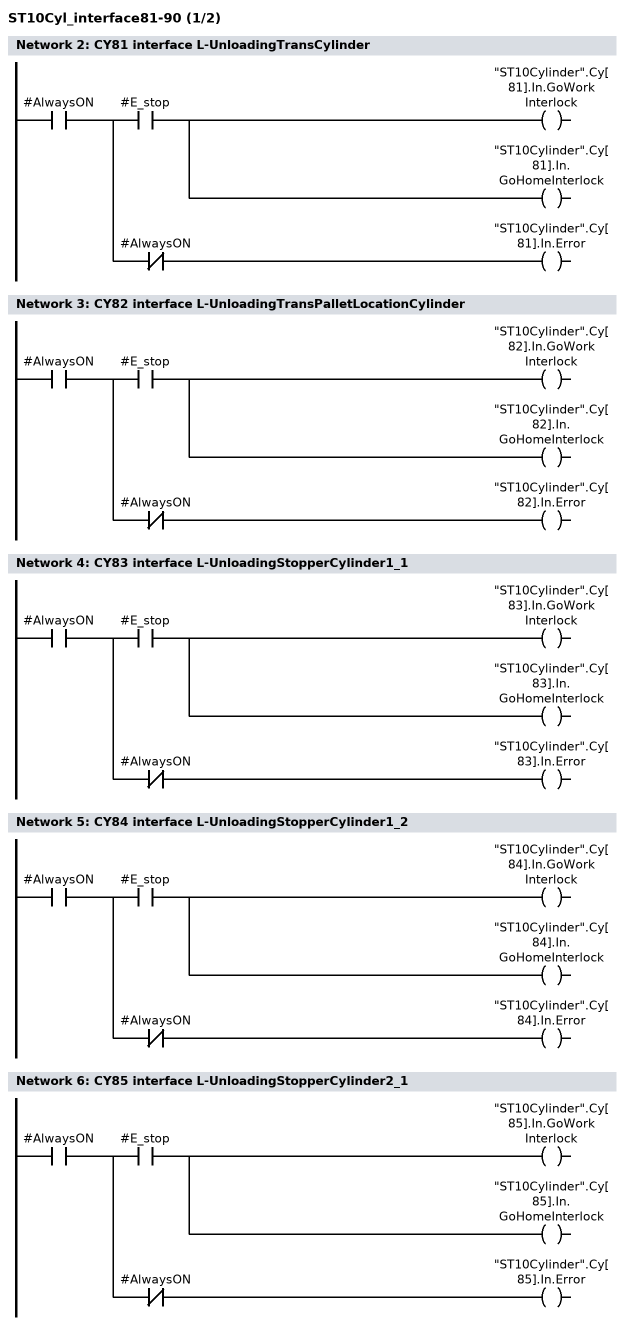
   RUNG wire#powerrail
      Contact( #AlwaysON )
      wire#w1
      Contact( #E_stop )
      wire#w2
      Coil( "ST10Cylinder".Cy[81].In.GoWorkInterlock )
   END_RUNG
   RUNG wire#w2
      Coil( "ST10Cylinder".Cy[81].In.GoHomeInterlock )
   END_RUNG
   RUNG wire#w1
      I_Contact( #AlwaysON )
      Coil( "ST10Cylinder".Cy[81].In.Error )
   END_RUNG
   // the same network as SCL:
   "ST10Cylinder".Cy[81].In.GoWorkInterlock := #AlwaysON AND #E_stop;
   "ST10Cylinder".Cy[81].In.GoHomeInterlock := #AlwaysON AND #E_stop;
   "ST10Cylinder".Cy[81].In.Error := #AlwaysON AND NOT #AlwaysON;
END_REGION

REGION Network 3: CY82 interface L-UnloadingTransPalletLocationCylinder
   RUNG wire#powerrail
      Contact( #AlwaysON )
      wire#w1
      Contact( #E_stop )
      wire#w2
      Coil( "ST10Cylinder".Cy[82].In.GoWorkInterlock )
   END_RUNG
   RUNG wire#w2
      Coil( "ST10Cylinder".Cy[82].In.GoHomeInterlock )
   END_RUNG
   RUNG wire#w1
      I_Contact( #AlwaysON )
      Coil( "ST10Cylinder".Cy[82].In.Error )
   END_RUNG
   // the same network as SCL:
   "ST10Cylinder".Cy[82].In.GoWorkInterlock := #AlwaysON AND #E_stop;
   "ST10Cylinder".Cy[82].In.GoHomeInterlock := #AlwaysON AND #E_stop;
   "ST10Cylinder".Cy[82].In.Error := #AlwaysON AND NOT #AlwaysON;
END_REGION

REGION Network 4: CY83 interface L-UnloadingStopperCylinder1_1
   RUNG wire#powerrail
      Contact( #AlwaysON )
      wire#w1
      Contact( #E_stop )
      wire#w2
      Coil( "ST10Cylinder".Cy[83].In.GoWorkInterlock )
   END_RUNG
   RUNG wire#w2
      Coil( "ST10Cylinder".Cy[83].In.GoHomeInterlock )
   END_RUNG
   RUNG wire#w1
      I_Contact( #AlwaysON )
      Coil( "ST10Cylinder".Cy[83].In.Error )
   END_RUNG
   // the same network as SCL:
   "ST10Cylinder".Cy[83].In.GoWorkInterlock := #AlwaysON AND #E_stop;
   "ST10Cylinder".Cy[83].In.GoHomeInterlock := #AlwaysON AND #E_stop;
   "ST10Cylinder".Cy[83].In.Error := #AlwaysON AND NOT #AlwaysON;
END_REGION

REGION Network 5: CY84 interface L-UnloadingStopperCylinder1_2
   RUNG wire#powerrail
      Contact( #AlwaysON )
      wire#w1
      Contact( #E_stop )
      wire#w2
      Coil( "ST10Cylinder".Cy[84].In.GoWorkInterlock )
   END_RUNG
   RUNG wire#w2
      Coil( "ST10Cylinder".Cy[84].In.GoHomeInterlock )
   END_RUNG
   RUNG wire#w1
      I_Contact( #AlwaysON )
      Coil( "ST10Cylinder".Cy[84].In.Error )
   END_RUNG
   // the same network as SCL:
   "ST10Cylinder".Cy[84].In.GoWorkInterlock := #AlwaysON AND #E_stop;
   "ST10Cylinder".Cy[84].In.GoHomeInterlock := #AlwaysON AND #E_stop;
   "ST10Cylinder".Cy[84].In.Error := #AlwaysON AND NOT #AlwaysON;
END_REGION

REGION Network 6: CY85 interface L-UnloadingStopperCylinder2_1
   RUNG wire#powerrail
      Contact( #AlwaysON )
      wire#w1
      Contact( #E_stop )
      wire#w2
      Coil( "ST10Cylinder".Cy[85].In.GoWorkInterlock )
   END_RUNG
   RUNG wire#w2
      Coil( "ST10Cylinder".Cy[85].In.GoHomeInterlock )
   END_RUNG
   RUNG wire#w1
      I_Contact( #AlwaysON )
      Coil( "ST10Cylinder".Cy[85].In.Error )
   END_RUNG
   // the same network as SCL:
   "ST10Cylinder".Cy[85].In.GoWorkInterlock := #AlwaysON AND #E_stop;
   "ST10Cylinder".Cy[85].In.GoHomeInterlock := #AlwaysON AND #E_stop;
   "ST10Cylinder".Cy[85].In.Error := #AlwaysON AND NOT #AlwaysON;
END_REGION

REGION Network 7: CY86 interface L-UnloadingStopperCylinder2_2
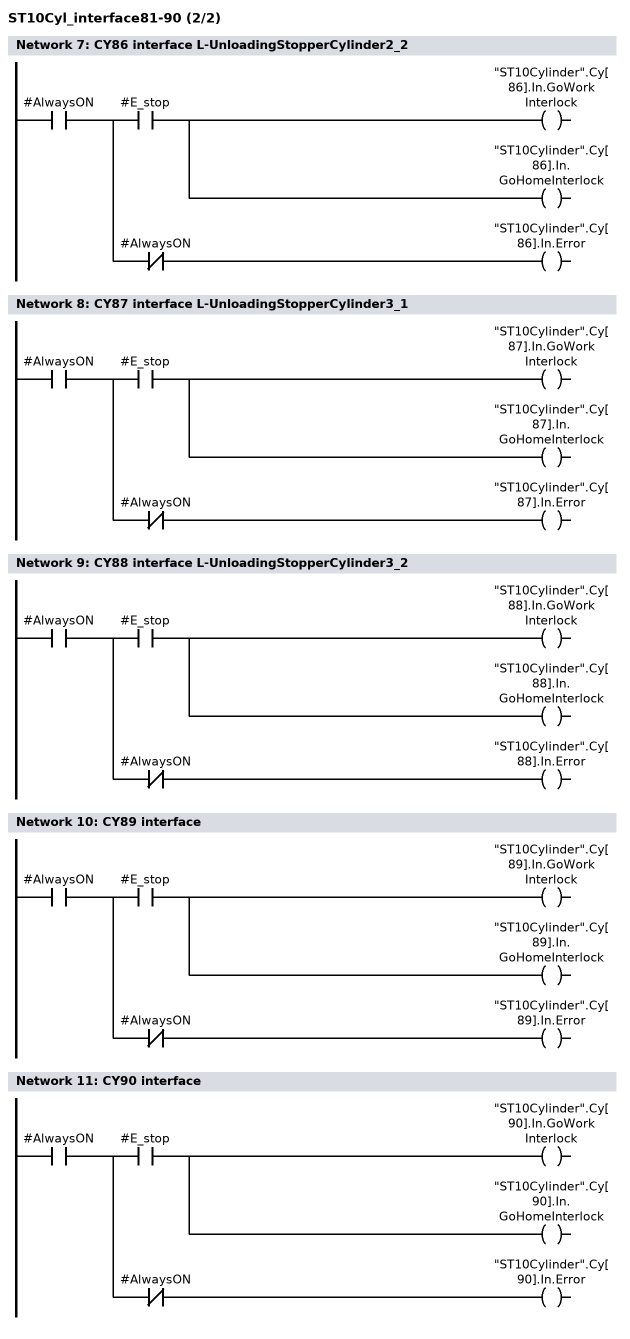
   RUNG wire#powerrail
      Contact( #AlwaysON )
      wire#w1
      Contact( #E_stop )
      wire#w2
      Coil( "ST10Cylinder".Cy[86].In.GoWorkInterlock )
   END_RUNG
   RUNG wire#w2
      Coil( "ST10Cylinder".Cy[86].In.GoHomeInterlock )
   END_RUNG
   RUNG wire#w1
      I_Contact( #AlwaysON )
      Coil( "ST10Cylinder".Cy[86].In.Error )
   END_RUNG
   // the same network as SCL:
   "ST10Cylinder".Cy[86].In.GoWorkInterlock := #AlwaysON AND #E_stop;
   "ST10Cylinder".Cy[86].In.GoHomeInterlock := #AlwaysON AND #E_stop;
   "ST10Cylinder".Cy[86].In.Error := #AlwaysON AND NOT #AlwaysON;
END_REGION

REGION Network 8: CY87 interface L-UnloadingStopperCylinder3_1
   RUNG wire#powerrail
      Contact( #AlwaysON )
      wire#w1
      Contact( #E_stop )
      wire#w2
      Coil( "ST10Cylinder".Cy[87].In.GoWorkInterlock )
   END_RUNG
   RUNG wire#w2
      Coil( "ST10Cylinder".Cy[87].In.GoHomeInterlock )
   END_RUNG
   RUNG wire#w1
      I_Contact( #AlwaysON )
      Coil( "ST10Cylinder".Cy[87].In.Error )
   END_RUNG
   // the same network as SCL:
   "ST10Cylinder".Cy[87].In.GoWorkInterlock := #AlwaysON AND #E_stop;
   "ST10Cylinder".Cy[87].In.GoHomeInterlock := #AlwaysON AND #E_stop;
   "ST10Cylinder".Cy[87].In.Error := #AlwaysON AND NOT #AlwaysON;
END_REGION

REGION Network 9: CY88 interface L-UnloadingStopperCylinder3_2
   RUNG wire#powerrail
      Contact( #AlwaysON )
      wire#w1
      Contact( #E_stop )
      wire#w2
      Coil( "ST10Cylinder".Cy[88].In.GoWorkInterlock )
   END_RUNG
   RUNG wire#w2
      Coil( "ST10Cylinder".Cy[88].In.GoHomeInterlock )
   END_RUNG
   RUNG wire#w1
      I_Contact( #AlwaysON )
      Coil( "ST10Cylinder".Cy[88].In.Error )
   END_RUNG
   // the same network as SCL:
   "ST10Cylinder".Cy[88].In.GoWorkInterlock := #AlwaysON AND #E_stop;
   "ST10Cylinder".Cy[88].In.GoHomeInterlock := #AlwaysON AND #E_stop;
   "ST10Cylinder".Cy[88].In.Error := #AlwaysON AND NOT #AlwaysON;
END_REGION

REGION Network 10: CY89 interface
   RUNG wire#powerrail
      Contact( #AlwaysON )
      wire#w1
      Contact( #E_stop )
      wire#w2
      Coil( "ST10Cylinder".Cy[89].In.GoWorkInterlock )
   END_RUNG
   RUNG wire#w2
      Coil( "ST10Cylinder".Cy[89].In.GoHomeInterlock )
   END_RUNG
   RUNG wire#w1
      I_Contact( #AlwaysON )
      Coil( "ST10Cylinder".Cy[89].In.Error )
   END_RUNG
   // the same network as SCL:
   "ST10Cylinder".Cy[89].In.GoWorkInterlock := #AlwaysON AND #E_stop;
   "ST10Cylinder".Cy[89].In.GoHomeInterlock := #AlwaysON AND #E_stop;
   "ST10Cylinder".Cy[89].In.Error := #AlwaysON AND NOT #AlwaysON;
END_REGION

REGION Network 11: CY90 interface
   RUNG wire#powerrail
      Contact( #AlwaysON )
      wire#w1
      Contact( #E_stop )
      wire#w2
      Coil( "ST10Cylinder".Cy[90].In.GoWorkInterlock )
   END_RUNG
   RUNG wire#w2
      Coil( "ST10Cylinder".Cy[90].In.GoHomeInterlock )
   END_RUNG
   RUNG wire#w1
      I_Contact( #AlwaysON )
      Coil( "ST10Cylinder".Cy[90].In.Error )
   END_RUNG
   // the same network as SCL:
   "ST10Cylinder".Cy[90].In.GoWorkInterlock := #AlwaysON AND #E_stop;
   "ST10Cylinder".Cy[90].In.GoHomeInterlock := #AlwaysON AND #E_stop;
   "ST10Cylinder".Cy[90].In.Error := #AlwaysON AND NOT #AlwaysON;
END_REGION
END_FUNCTION

FUNCTION "ST10_ChangeOver" : Void   // FC1008, LAD
{ S7_Optimized_Access := 'FALSE' }
// stored: AutoNumber false, SetENOAutomatically false
   VAR_TEMP
      sString : String[50];
      FixtureNumber : Int;
      FixtureIndex : Int;
      tRET_VAL : Int;
   END_VAR
BEGIN

REGION Network 1: Recipe Active
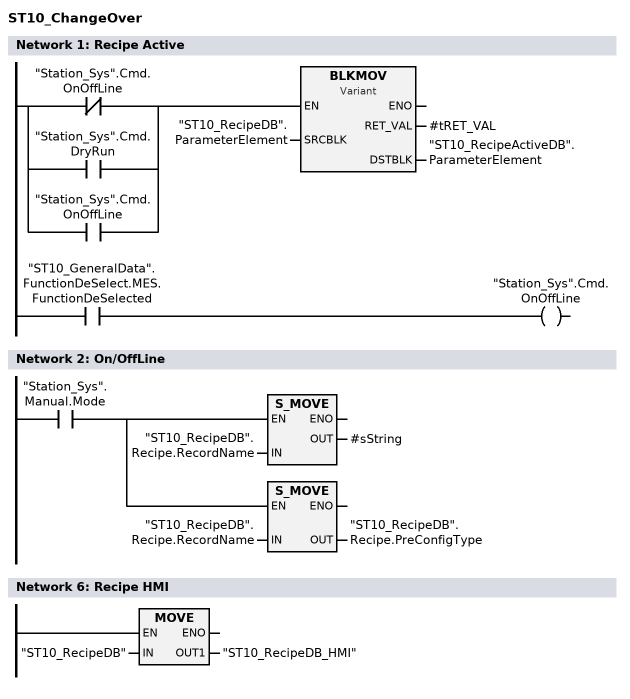
   RUNG wire#powerrail
      I_Contact( "Station_Sys".Cmd.OnOffLine )
      wire#w1
      { S7_Templates := "blk_type := Variant" } BLKMOV(SRCBLK := "ST10_RecipeDB".ParameterElement, RET_VAL => #tRET_VAL, DSTBLK => "ST10_RecipeActiveDB".ParameterElement)
   END_RUNG
   RUNG wire#powerrail
      Contact( "Station_Sys".Cmd.DryRun )
   END_RUNG wire#w1
   RUNG wire#powerrail
      Contact( "Station_Sys".Cmd.OnOffLine )
   END_RUNG wire#w1
   RUNG wire#powerrail
      Contact( "ST10_GeneralData".FunctionDeSelect.MES.FunctionDeSelected )
      Coil( "Station_Sys".Cmd.OnOffLine )
   END_RUNG
   // the same network as SCL:
   IF NOT "Station_Sys".Cmd.OnOffLine OR "Station_Sys".Cmd.DryRun OR "Station_Sys".Cmd.OnOffLine THEN
       #tRET_VAL := BLKMOV(SRCBLK := "ST10_RecipeDB".ParameterElement,
                           DSTBLK => "ST10_RecipeActiveDB".ParameterElement);
   END_IF;
   "Station_Sys".Cmd.OnOffLine := "ST10_GeneralData".FunctionDeSelect.MES.FunctionDeSelected;
END_REGION

REGION Network 2: On/OffLine
   RUNG wire#powerrail
      Contact( "Station_Sys".Manual.Mode )
      wire#w1
      S_Move(in := "ST10_RecipeDB".Recipe.RecordName, out => #sString)
   END_RUNG
   RUNG wire#w1
      S_Move(in := "ST10_RecipeDB".Recipe.RecordName, out => "ST10_RecipeDB".Recipe.PreConfigType)
   END_RUNG
   // the same network as SCL:
   IF "Station_Sys".Manual.Mode THEN
       #sString := "ST10_RecipeDB".Recipe.RecordName;
       "ST10_RecipeDB".Recipe.PreConfigType := "ST10_RecipeDB".Recipe.RecordName;
   END_IF;
END_REGION

NETWORK
TITLE = 换型功能块调用 / Transposition function block call
//"ST10_RecipeDB".Recipe.PreConfigType    AUTO CONFIG, When PLC activate change over, Set Recipe data record Tags
//"ST10_RecipeDB".ParameterElement.TypeName    HMI MANUAL CONFIG, HMI Recipe data record element:Product_type
//HMI Recipe data record element Product_type set value must be same with HMI Recipe data record Name

      A     "ChangeOver_DB".Global.ChangeOverActive;
      A     "Station_Sys".Auto.Mode;
      =     "ST10_RecipeDB".Recipe.Trigger;

      CALL  "ChangeOver"
      ( iCheckType      := "ST10_RecipeDB".ParameterElement.TypeName,
        "iPulse*500ms"  := "Sys".COM.FlashTime500mS,
        iReset          := "Station_Sys".Cmd.Reset,
        Ret_Val         := "ST10_RecipeDB".Recipe.Ret,
        oPulse          := "ST10_RecipeDB".Recipe.Pulse,
        oEqual          := "ST10_RecipeDB".Recipe.Equal,  // CheckType=PreConfigType, indicate ChangerOver successfully
        ioPreConfigType := "ST10_RecipeDB".Recipe.PreConfigType,
        ioCurrentName   := "ST10_RecipeDB".Recipe.RecordName,
        iotime          := "ST10_RecipeDB".Recipe."time",
        ioTrigger       := "ST10_RecipeDB".Recipe.Trigger,
        ioPosEdg        := "ST10_RecipeDB".Recipe.PosEdg,
        ioAlarm         := "ST10_RecipeDB".Recipe.Alarm,
        ioPls           := "ST10_RecipeDB".Recipe.Pls
      );




REGION Network 4 (SCL): Fixture换型工装 / Fixture Changing fixture
   //Fixture 1 输入轴换型X轴工装
   //工装检测屏蔽条件
   "ST10_GeneralData".FixtureIDCheck[1].FixtureCheckUnEnable := 0;

   //工装检测传感器赋值

   "ST10_GeneralData".FixtureIDCheck[1].FixtureIDCheckValue.%X0 := 0;
   "ST10_GeneralData".FixtureIDCheck[1].FixtureIDCheckValue.%X1 := 0;
   "ST10_GeneralData".FixtureIDCheck[1].FixtureIDCheckValue.%X2 := 0;
   "ST10_GeneralData".FixtureIDCheck[1].FixtureIDCheckValue.%X3 := 0;
   "ST10_GeneralData".FixtureIDCheck[1].FixtureIDCheckValue.%X4 := 0;
   "ST10_GeneralData".FixtureIDCheck[1].FixtureIDCheckValue.%X5 := 0;
   "ST10_GeneralData".FixtureIDCheck[1].FixtureIDCheckValue.%X6 := 0;
   "ST10_GeneralData".FixtureIDCheck[1].FixtureIDCheckValue.%X7 := 0;
END_REGION

REGION Network 5 (SCL): FixtureID Check Call
   //循环数量为工装检测的数量

   #FixtureNumber := 1;

   //工装检测功能块调用

   #FixtureIndex := 1;

   FOR #FixtureIndex := 1 TO #FixtureNumber DO

       "fcFixtureCheck"(iRecipeSetValue := "ST10_RecipeDB".ParameterElement.FixtureID[#FixtureIndex],
                        FixtureIDCheck := "ST10_GeneralData".FixtureIDCheck[#FixtureIndex]);

   END_FOR;
END_REGION

REGION Network 6: Recipe HMI
   RUNG wire#powerrail
      Move(in := "ST10_RecipeDB", out1 => "ST10_RecipeDB_HMI")
   END_RUNG
   // the same network as SCL:
   "ST10_RecipeDB_HMI" := "ST10_RecipeDB";
END_REGION
END_FUNCTION

FUNCTION "ChangeOver" : Bool   // FC3002, SCL
TITLE = ChangeOverV3
{ S7_Optimized_Access := 'FALSE' }
AUTHOR : STD
FAMILY : RCS
VERSION : 18.0
// stored: AutoNumber false, SetENOAutomatically true
   VAR_INPUT
      iCheckType : String;   // Person Confirm input type ID/NAME
      "iPulse*500ms" : Bool;   // pulse
      iReset : Bool;
   END_VAR
   VAR_OUTPUT
      oPulse : Bool;   // system pulse[HMI Variable Must keep continous mode]
      oEqual : Bool;
   END_VAR
   VAR_IN_OUT
      ioPreConfigType : String;   // to be changed recipe ID/NAME
      ioCurrentName : String;   // current recipe record name
      iotime : Int;   // time record
      ioTrigger : Bool;   // trigger for changeing over
      ioPosEdg : Bool;   // postive edge bit
      ioAlarm : Bool;   // Changover time out
      ioPls : Bool;
   END_VAR
   VAR_TEMP
      tpPosEdg : Bool;
      tpPls : Bool;
   END_VAR
   // Ret_Val : 0-NG/1-OK
BEGIN
   //---------------------------------------------------------------//
   //FunctionName:ChangeOverV3
   //FunctionDescription:ChangeOver
   //---------------------------------------------------------------//
   (*in:

   iPreConfigType  String
   iLastType   String
   iPulse*500ms    Bool
   iTrigger    Bool


   //inout:
   //out:
   oPulse  Bool
   oAlarm  Bool

   *)
   //---------------------------------------------------------------//
   //Version:V2
   //D&T:2016-11-125
   //Group:RCS
   //Author:JM
   //-------------------------Modify1----------------------------------//
   //Version:V3.0
   //D&T:2016-11-28
   //Group: RCS
   //Author:JM
   //Modify: add timeout bit 
   //-------------------------Modify2----------------------------------//
   //Version:V3.0
   //D&T:20180416
   //Group: RCS
   //Author:JM
   //Modify:
   // Add pls flag in order to keep paramter that download after modifier safe.
   #tpPls := #ioTrigger AND NOT #ioPls;
   #ioPls := #ioTrigger;
   #tpPosEdg := #"iPulse*500ms" AND NOT #ioPosEdg;
   #ioPosEdg := #"iPulse*500ms";
   #oEqual := #ioPreConfigType = #iCheckType AND #ioPreConfigType<>'';


   // IF #tpPls THEN
   //     #ioPreConfigType:='';
   // END_IF;
   IF (#iReset AND #ioAlarm) OR #oEqual THEN
       #ioAlarm := 0;
   END_IF;
   IF NOT #ioTrigger THEN
       #ChangeOver := 0;
       #iotime := 0;
       // #oAlarm := 0;
       RETURN;
   ELSE
       IF #tpPosEdg THEN
           #iotime := #iotime + 1;
       END_IF;
       IF #iotime >= 10 THEN
           #ioAlarm := 1;
           #ioTrigger := 0;
           // ELSE
           //     #oAlarm := 0;
       END_IF;
       #ChangeOver := 0;
       // #tpCurrentProductlen := LEN(#tpCurrentProduct);
       // #tpLastProductlen := LEN(#tpLastProduct);
       IF #ioPreConfigType <> #iCheckType THEN
           #oPulse := #"iPulse*500ms";
           RETURN;
       ELSE
           IF #ioCurrentName <> #ioPreConfigType THEN
               #ioCurrentName := #ioPreConfigType;
           END_IF;
           #iotime := 0;
           #ioAlarm := 0;
           #oPulse := 0;
           #ChangeOver := 1;
           #ioTrigger := 0;
           ENO := 1;
       END_IF;

   END_IF;
END_FUNCTION

FUNCTION "ST10_Device" : Void   // FC1010, LAD
{ S7_Optimized_Access := 'TRUE' }
// stored: AutoNumber false, SetENOAutomatically false
   VAR_INPUT
      iSysMode : "RCS_SysComInterface_V1";
   END_VAR
BEGIN

NETWORK
TITLE = SafetyGate

      CALL  "ST10_SafetyGate"
      ( iSysMode := #iSysMode
      );


NETWORK
TITLE = PartData

      CALL  "ST10_PartData"
      ( iSysMode := #iSysMode
      );


NETWORK
TITLE = Analog

      CALL  "ST10_Analog"
      ( iSysMode := #iSysMode
      );


REGION Network 4: SR Scan
END_REGION

REGION Network 7: CuringOven
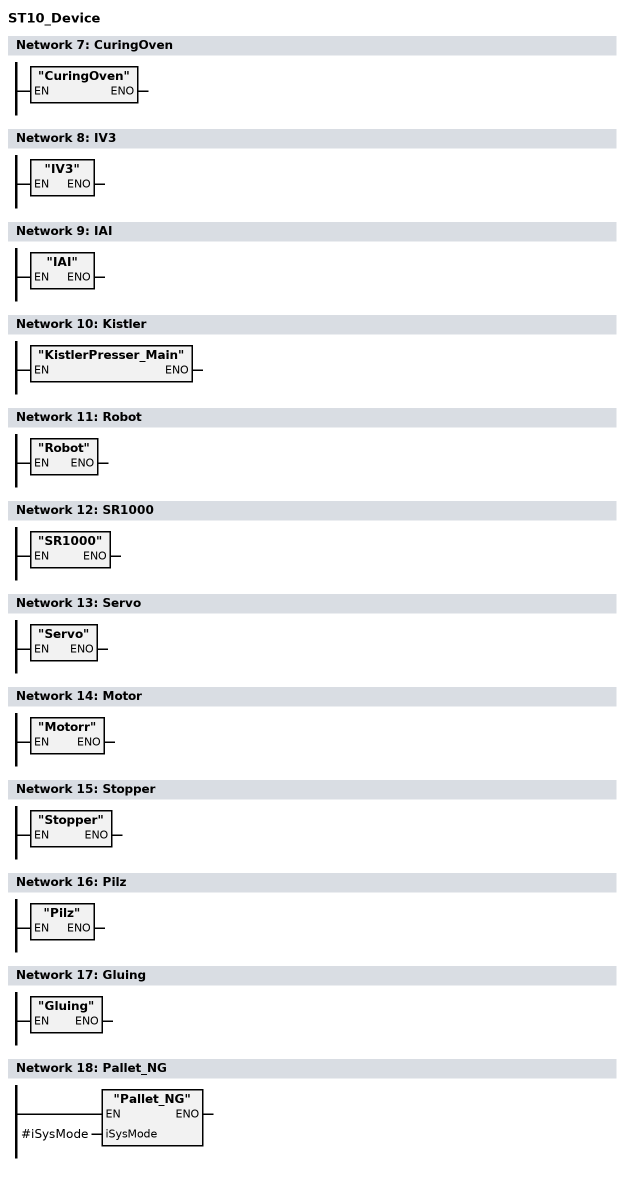
   RUNG wire#powerrail
      "CuringOven"()
   END_RUNG
   // the same network as SCL:
   "CuringOven"();
END_REGION

REGION Network 8: IV3
   RUNG wire#powerrail
      "IV3"()
   END_RUNG
   // the same network as SCL:
   "IV3"();
END_REGION

REGION Network 9: IAI
   RUNG wire#powerrail
      "IAI"()
   END_RUNG
   // the same network as SCL:
   "IAI"();
END_REGION

REGION Network 10: Kistler
   RUNG wire#powerrail
      "KistlerPresser_Main"()
   END_RUNG
   // the same network as SCL:
   "KistlerPresser_Main"();
END_REGION

REGION Network 11: Robot
   RUNG wire#powerrail
      "Robot"()
   END_RUNG
   // the same network as SCL:
   "Robot"();
END_REGION

REGION Network 12: SR1000
   RUNG wire#powerrail
      "SR1000"()
   END_RUNG
   // the same network as SCL:
   "SR1000"();
END_REGION

REGION Network 13: Servo
   RUNG wire#powerrail
      "Servo"()
   END_RUNG
   // the same network as SCL:
   "Servo"();
END_REGION

REGION Network 14: Motor
   RUNG wire#powerrail
      "Motorr"()
   END_RUNG
   // the same network as SCL:
   "Motorr"();
END_REGION

REGION Network 15: Stopper
   RUNG wire#powerrail
      "Stopper"()
   END_RUNG
   // the same network as SCL:
   "Stopper"();
END_REGION

REGION Network 16: Pilz
   RUNG wire#powerrail
      "Pilz"()
   END_RUNG
   // the same network as SCL:
   "Pilz"();
END_REGION

REGION Network 17: Gluing
   RUNG wire#powerrail
      "Gluing"()
   END_RUNG
   // the same network as SCL:
   "Gluing"();
END_REGION

REGION Network 18: Pallet_NG
   RUNG wire#powerrail
      "Pallet_NG"(iSysMode := #iSysMode)
   END_RUNG
   // the same network as SCL:
   "Pallet_NG"(iSysMode := #iSysMode);
END_REGION
END_FUNCTION

FUNCTION "ST10_SafetyGate" : Void   // FC1140, SCL
{ S7_Optimized_Access := 'TRUE' }
// stored: AutoNumber false, SetENOAutomatically false
   VAR_INPUT
      iSysMode : "RCS_SysComInterface_V1";
   END_VAR
   VAR_TEMP
      idex : Int;
   END_VAR
BEGIN


   REGION SafetyGate 1    
       //定义编号
       #idex := 1;
       //功能块调用
       //
       "ST10_SafetyGate1_DB"(iSysInface := #iSysMode,
                             "iSafetyGate Opened Monitor" := NOT "iSafety door Locking FeedBack_1",
                             "iSafetyGate Locked Monitor" := "ST10_SysOutput".SafetyDoorCoil[1],
                             i1s_Pulse := "ClockMemory1s",
                             iMode :=1,
                              "oSafetyGate LockedLamp"=>"ST10_SafetyGate_InterfaceDB" .SafetyDoorLamp[1],
                              ioSafetyGateLock := "ST10_SysOutput".SafetyDoorCoil[1],
                              ioHMI_Interface := "ST10_SafetyGate_InterfaceDB".aDev[#idex]);

   END_REGION

   REGION SafetyGate 2    
       //定义编号
       #idex := 2;
       //功能块调用
       //
       "ST10_SafetyGate2_DB"(iSysInface := #iSysMode,
                             "iSafetyGate Opened Monitor" := NOT "iSafety door Locking FeedBack_2",
                             "iSafetyGate Locked Monitor" := "ST10_SysOutput".SafetyDoorCoil[2],
                             i1s_Pulse := "ClockMemory1s",
                             iMode :=1,
                              "oSafetyGate LockedLamp"=> "ST10_SafetyGate_InterfaceDB" .SafetyDoorLamp[2],
                              ioSafetyGateLock := "ST10_SysOutput".SafetyDoorCoil[2],
                              ioHMI_Interface := "ST10_SafetyGate_InterfaceDB".aDev[#idex]);

   END_REGION

   REGION SafetyGate 3    
       //定义编号
       #idex := 3;
       //功能块调用
       //
       "ST10_SafetyGate3_DB"(iSysInface := #iSysMode,
                             "iSafetyGate Opened Monitor" := NOT "iSafety door Locking FeedBack_3",
                             "iSafetyGate Locked Monitor" := "ST10_SysOutput".SafetyDoorCoil[3],
                             i1s_Pulse := "ClockMemory1s",
                             iMode :=1,
                              "oSafetyGate LockedLamp"=> "ST10_SafetyGate_InterfaceDB" .SafetyDoorLamp[3],
                              ioSafetyGateLock := "ST10_SysOutput".SafetyDoorCoil[3],
                              ioHMI_Interface := "ST10_SafetyGate_InterfaceDB".aDev[#idex]);

   END_REGION

   REGION SafetyGate 4    
       //定义编号
       #idex := 4;
       //功能块调用
       //
       "ST10_SafetyGate4_DB"(iSysInface := #iSysMode,
                              "iSafetyGate Opened Monitor" := NOT "iSafety door Locking FeedBack_4",
                              "iSafetyGate Locked Monitor" := "ST10_SysOutput".SafetyDoorCoil[4],
                              i1s_Pulse := "ClockMemory1s",
                              iMode :=1,
                              "oSafetyGate LockedLamp"=>"ST10_SafetyGate_InterfaceDB" .SafetyDoorLamp[4],
                              ioSafetyGateLock := "ST10_SysOutput".SafetyDoorCoil[4],
                              ioHMI_Interface := "ST10_SafetyGate_InterfaceDB".aDev[#idex]);

   END_REGION

   REGION SafetyGate 5    
       //定义编号
       #idex := 5;
       //功能块调用
       //
       "ST10_SafetyGate5_DB"(iSysInface := #iSysMode,
                             "iSafetyGate Opened Monitor" := NOT "iSafety door Locking FeedBack_5",
                             "iSafetyGate Locked Monitor" := "ST10_SysOutput".SafetyDoorCoil[5],
                             i1s_Pulse := "ClockMemory1s",
                             iMode :=1,
                             "oSafetyGate LockedLamp" => "ST10_SafetyGate_InterfaceDB".SafetyDoorLamp[5],
                             ioSafetyGateLock := "ST10_SysOutput".SafetyDoorCoil[5],
                             ioHMI_Interface := "ST10_SafetyGate_InterfaceDB".aDev[#idex]);

   END_REGION

   REGION SafetyGate 6    
       //定义编号
       #idex := 6;
       //功能块调用
       //
       "ST10_SafetyGate6_DB"(iSysInface := #iSysMode,
                             "iSafetyGate Opened Monitor" := NOT "iSafety door Locking FeedBack_6",
                             "iSafetyGate Locked Monitor" := "ST10_SysOutput".SafetyDoorCoil[6],
                             i1s_Pulse := "ClockMemory1s",
                             iMode :=1,
                             "oSafetyGate LockedLamp" => "ST10_SafetyGate_InterfaceDB".SafetyDoorLamp[6],
                             ioSafetyGateLock := "ST10_SysOutput".SafetyDoorCoil[6],
                             ioHMI_Interface := "ST10_SafetyGate_InterfaceDB".aDev[#idex]);

                          END_REGION

   REGION SafetyGate 7    
       //定义编号
       #idex := 7;
       //功能块调用
       //
       "ST10_SafetyGate7_DB"(iSysInface := #iSysMode,
                             "iSafetyGate Opened Monitor" := NOT "iSafety door Locking FeedBack_7",
                             "iSafetyGate Locked Monitor" := "ST10_SysOutput".SafetyDoorCoil[7],
                             i1s_Pulse := "ClockMemory1s",
                             iMode :=1,
                             "oSafetyGate LockedLamp" => "ST10_SafetyGate_InterfaceDB".SafetyDoorLamp[7],
                             ioSafetyGateLock := "ST10_SysOutput".SafetyDoorCoil[7],
                             ioHMI_Interface := "ST10_SafetyGate_InterfaceDB".aDev[#idex]);

   END_REGION

   REGION SafetyGate 8    
       //定义编号
       #idex := 8;
       //功能块调用
       //
       "ST10_SafetyGate8_DB"(iSysInface := #iSysMode,
                             "iSafetyGate Opened Monitor" := NOT "iSafety door Locking FeedBack_8",
                             "iSafetyGate Locked Monitor" := "ST10_SysOutput".SafetyDoorCoil[8],
                             i1s_Pulse := "ClockMemory1s",
                             iMode :=1,
                             "oSafetyGate LockedLamp" => "ST10_SafetyGate_InterfaceDB".SafetyDoorLamp[8],
                             ioSafetyGateLock := "ST10_SysOutput".SafetyDoorCoil[8],
                             ioHMI_Interface := "ST10_SafetyGate_InterfaceDB".aDev[#idex]);

                          END_REGION

   REGION SafetyGate 9    
    //定义编号
     #idex := 9;
    //功能块调用
    //
      "ST10_SafetyGate9_DB"(iSysInface := #iSysMode,
                            "iSafetyGate Opened Monitor" := NOT "iSafety Door Locking FeedBack",
                           "iSafetyGate Locked Monitor" := "ST10_SysOutput".SafetyDoorCoil[9],
                           i1s_Pulse := "ClockMemory1s",
                           iMode :=1,
                            "oSafetyGate LockedLamp" => "ST10_SafetyGate_InterfaceDB".SafetyDoorLamp[9],
                            ioSafetyGateLock := "ST10_SysOutput".SafetyDoorCoil[9],
                            ioHMI_Interface := "ST10_SafetyGate_InterfaceDB".aDev[#idex]);

   END_REGION

   REGION SafetyGate 11    
    //定义编号
   #idex := 11;
   //功能块调用
   //
   "ST10_MaterialGate1_DB"(iSysInface := #iSysMode,
                           "iSafetyGate Opened Monitor" := NOT "iMateriel Door Locking FeedBack_H1",
                          "iSafetyGate Locked Monitor" := "ST10_SysOutput".MaterialDoorCoil[1],
                          i1s_Pulse := "ClockMemory1s",
                          iMode :=2,
                            "oSafetyGate LockedLamp" => "ST10_SafetyGate_InterfaceDB".SafetyDoorLamp[11],
                            ioSafetyGateLock := "ST10_SysOutput".MaterialDoorCoil[1],
                            ioHMI_Interface := "ST10_SafetyGate_InterfaceDB".aDev[#idex]);

   END_REGION

   REGION SafetyGate 12    
       //定义编号
       #idex := 12;
       //功能块调用
       //
       "ST10_MaterialGate2_DB"(iSysInface := #iSysMode,
                               "iSafetyGate Opened Monitor" := NOT "iMateriel Door Locking FeedBack_H2",
                             "iSafetyGate Locked Monitor" := "ST10_SysOutput".MaterialDoorCoil[2],
                             i1s_Pulse := "ClockMemory1s",
                             iMode :=2,
                             "oSafetyGate LockedLamp" => "ST10_SafetyGate_InterfaceDB".SafetyDoorLamp[12],
                             ioSafetyGateLock := "ST10_SysOutput".MaterialDoorCoil[2],
                             ioHMI_Interface := "ST10_SafetyGate_InterfaceDB".aDev[#idex]);

   END_REGION

   REGION SafetyGate 13    
       //定义编号
       #idex := 13;
       //功能块调用
       //
       "ST10_MaterialGate3_DB"(iSysInface := #iSysMode,
                               "iSafetyGate Opened Monitor" := NOT "iMateriel Door Locking FeedBack_J1",
                             "iSafetyGate Locked Monitor" := "ST10_SysOutput".MaterialDoorCoil[3],
                             i1s_Pulse := "ClockMemory1s",
                             iMode :=2,
                             "oSafetyGate LockedLamp" => "ST10_SafetyGate_InterfaceDB".SafetyDoorLamp[13],
                             ioSafetyGateLock := "ST10_SysOutput".MaterialDoorCoil[3],
                             ioHMI_Interface := "ST10_SafetyGate_InterfaceDB".aDev[#idex]);

   END_REGION

   REGION SafetyGate 14    
       //定义编号
       #idex := 14;
       //功能块调用
       //
       "ST10_MaterialGate4_DB"(iSysInface := #iSysMode,
                               "iSafetyGate Opened Monitor" := NOT "iMateriel Door Locking FeedBack_J2",
                             "iSafetyGate Locked Monitor" := "ST10_SysOutput".MaterialDoorCoil[4],
                             i1s_Pulse := "ClockMemory1s",
                             iMode :=2,
                             "oSafetyGate LockedLamp" => "ST10_SafetyGate_InterfaceDB".SafetyDoorLamp[14],
                             ioSafetyGateLock := "ST10_SysOutput".MaterialDoorCoil[4],
                             ioHMI_Interface := "ST10_SafetyGate_InterfaceDB".aDev[#idex]);

   END_REGION

   REGION SafetyGate 15    
       //定义编号
       #idex := 15;
       //功能块调用
       //
       "ST10_MaterialGate5_DB"(iSysInface := #iSysMode,
                               "iSafetyGate Opened Monitor" := NOT "iMateriel Door Locking FeedBack_K1",
                             "iSafetyGate Locked Monitor" := "ST10_SysOutput".MaterialDoorCoil[5],
                             i1s_Pulse := "ClockMemory1s",
                             iMode :=2,
                             "oSafetyGate LockedLamp" => "ST10_SafetyGate_InterfaceDB".SafetyDoorLamp[15],
                             ioSafetyGateLock := "ST10_SysOutput".MaterialDoorCoil[5],
                             ioHMI_Interface := "ST10_SafetyGate_InterfaceDB".aDev[#idex]);

   END_REGION

   REGION SafetyGate 16    
       //定义编号
       #idex := 16;
       //功能块调用
       //
       "ST10_MaterialGate6_DB"(iSysInface := #iSysMode,
                               "iSafetyGate Opened Monitor" := NOT "iMateriel Door Locking FeedBack_K2",
                               "iSafetyGate Locked Monitor" := "ST10_SysOutput".MaterialDoorCoil[6],
                               i1s_Pulse := "ClockMemory1s",
                               iMode :=2,
                               "oSafetyGate LockedLamp" => "ST10_SafetyGate_InterfaceDB".SafetyDoorLamp[16],
                               ioSafetyGateLock := "ST10_SysOutput".MaterialDoorCoil[6],
                               ioHMI_Interface := "ST10_SafetyGate_InterfaceDB".aDev[#idex]);

   END_REGION

   REGION SafetyGate 17    
       //定义编号
       #idex := 17;
       //功能块调用
       //
       "ST10_MaterialGate7_DB"(iSysInface := #iSysMode,
                               "iSafetyGate Opened Monitor" := NOT "iMateriel Door Locking FeedBack_L1",
                               "iSafetyGate Locked Monitor" := "ST10_SysOutput".MaterialDoorCoil[7],
                               i1s_Pulse := "ClockMemory1s",
                               iMode :=2,
                             "oSafetyGate LockedLamp" => "ST10_SafetyGate_InterfaceDB".SafetyDoorLamp[17],
                             ioSafetyGateLock := "ST10_SysOutput".MaterialDoorCoil[7],
                             ioHMI_Interface := "ST10_SafetyGate_InterfaceDB".aDev[#idex]);

   END_REGION

   REGION SafetyGate 18    
       //定义编号
       #idex := 18;
       //功能块调用
       //
       "ST10_NGGate1_DB"(iSysInface := #iSysMode,
                         "iSafetyGate Opened Monitor" :=  "iE-NG-01 Safety Gate_Open",
                         "iSafetyGate Locked Monitor" := "iE-NG-01 Safety Gate_UnLock",
                               i1s_Pulse := "ClockMemory1s",
                               iMode := 2,
                               "oSafetyGate LockedLamp" => "ST10_SafetyGate_InterfaceDB".SafetyDoorLamp[18],
                               ioSafetyGateLock := "ST10_SysOutput".MaterialDoorCoil[8],
                               ioHMI_Interface := "ST10_SafetyGate_InterfaceDB".aDev[#idex]);

   END_REGION

   REGION SafetyGate 19    
       //定义编号
       #idex := 19;
       //功能块调用
       //
       "ST10_NGGate2_DB"(iSysInface := #iSysMode,
                         "iSafetyGate Opened Monitor" := "iE-NG-02 Safety Gate_Open",
                         "iSafetyGate Locked Monitor" := "iE-NG-02 Safety Gate_UnLock",
                         i1s_Pulse := "ClockMemory1s",
                         iMode := 2,
                         "oSafetyGate LockedLamp" => "ST10_SafetyGate_InterfaceDB".SafetyDoorLamp[19],
                         ioSafetyGateLock := "ST10_SysOutput".MaterialDoorCoil[9],
                         ioHMI_Interface := "ST10_SafetyGate_InterfaceDB".aDev[#idex]);

   END_REGION
END_FUNCTION

FUNCTION_BLOCK "SafetyGate"   // FB5200, LAD
{ S7_Optimized_Access := 'FALSE' }
VERSION : 0.1
// stored: AutoNumber false, IsIECCheckEnabled false, SetENOAutomatically false, UDAEnableTagReadback false
   VAR_INPUT
      iSysInface : "RCS_SysComInterface_V1";
      "iSafetyGate Opened Monitor" : Bool;   // 安全门打开状态监控
      "iSafetyGate Locked Monitor" : Bool;   // 安全门锁定状态监控
      i1s_Pulse : Bool;   // 1s脉冲信号
      "iSafetyGate AutoLock Timer" : Time := T#1s;   // 安全门自动模式下锁延时
      "iSafetyGate ManualLock Timer" : Time := T#60s;   // 安全门手动模式下锁定延时
      iMode : Int;
   END_VAR
   VAR_OUTPUT
      "oSafetyGate LockedLamp" { ExternalAccessible := 'False'; ExternalVisible := 'False'; ExternalWritable := 'False'} : Bool;   // 安全门解锁输出状态
   END_VAR
   VAR_IN_OUT
      ioSafetyGateLock : Bool;   // 安全门锁定输出
      ioHMI_Interface : "SafetyGateUDT";
   END_VAR
   VAR DB_SPECIFIC
      "sSafetyGate Timer" { S7_SetPoint := 'True'} : Array[1..5] of TON_TIME;
      sP_Trig : Array[1..10] of Bool;
      sN_Trig : Array[1..10] of Bool;
      "sSafetyGate UnlockRequest" { ExternalAccessible := 'False'; ExternalVisible := 'False'; ExternalWritable := 'False'} : Bool;   // 安全门开门请求标志位
      "sSafetyGate LockRequest" : Bool;
   END_VAR
   VAR_TEMP
      tAlyways_On : Bool;
      tAlyways_Off : Bool;
   END_VAR
   VAR_TEMP   // added for the SCL form of the ladder/FBD networks
      _w1 : Bool;
      _w2 : Bool;
      _w3 : Bool;
      _w4 : Bool;
      _w5 : Bool;
   END_VAR
BEGIN

REGION Network 1: #tAlyways_On
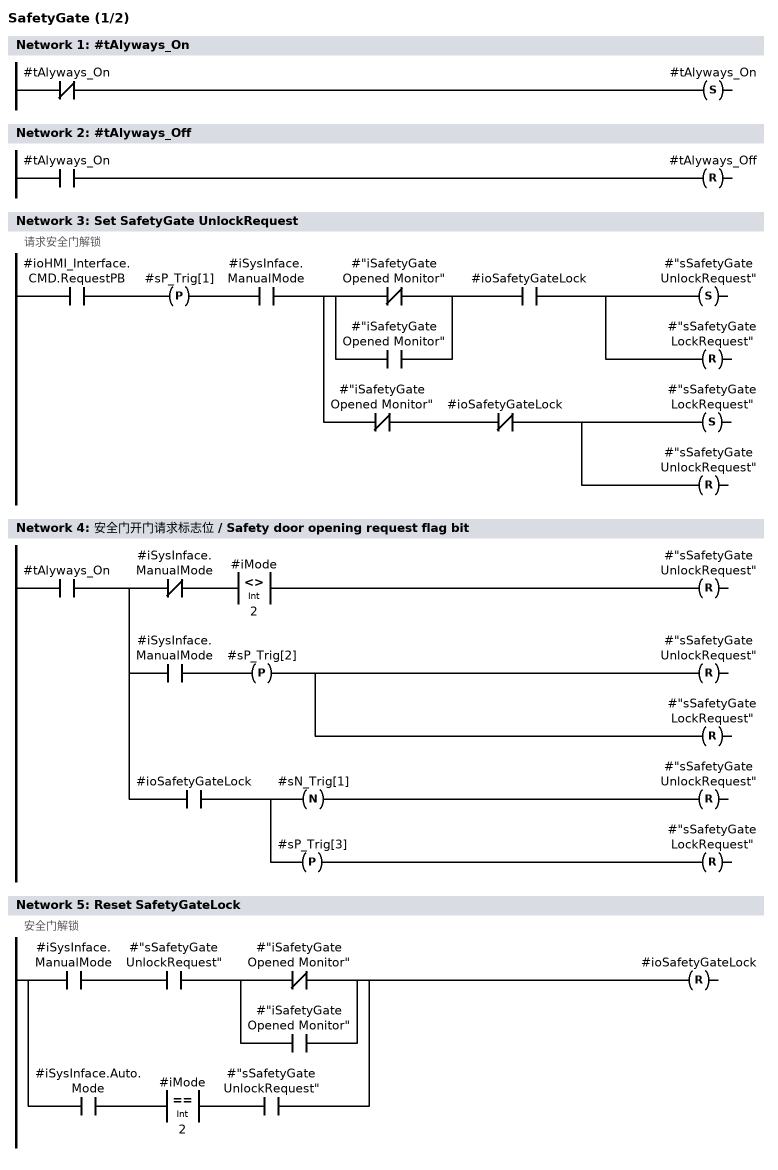
   RUNG wire#powerrail
      I_Contact( #tAlyways_On )
      S_Coil( #tAlyways_On )
   END_RUNG
   // the same network as SCL:
   IF NOT #tAlyways_On THEN #tAlyways_On := TRUE; END_IF;
END_REGION

REGION Network 2: #tAlyways_Off
   RUNG wire#powerrail
      Contact( #tAlyways_On )
      R_Coil( #tAlyways_Off )
   END_RUNG
   // the same network as SCL:
   IF #tAlyways_On THEN #tAlyways_Off := FALSE; END_IF;
END_REGION

REGION Network 3: Set SafetyGate UnlockRequest
   // 请求安全门解锁
   RUNG wire#powerrail
      Contact( #ioHMI_Interface.CMD.RequestPB )
      P_Trig( #sP_Trig[1] )
      Contact( #iSysInface.ManualMode )
      wire#w1
      I_Contact( #"iSafetyGate Opened Monitor" )
      wire#w2
      Contact( #ioSafetyGateLock )
      wire#w3
      S_Coil( #"sSafetyGate UnlockRequest" )
   END_RUNG
   RUNG wire#w1
      Contact( #"iSafetyGate Opened Monitor" )
   END_RUNG wire#w2
   RUNG wire#w3
      R_Coil( #"sSafetyGate LockRequest" )
   END_RUNG
   RUNG wire#w1
      I_Contact( #"iSafetyGate Opened Monitor" )
      I_Contact( #ioSafetyGateLock )
      wire#w4
      S_Coil( #"sSafetyGate LockRequest" )
   END_RUNG
   RUNG wire#w4
      R_Coil( #"sSafetyGate UnlockRequest" )
   END_RUNG
   // the same network as SCL:
   #_w1 := #ioHMI_Interface.CMD.RequestPB AND NOT #sP_Trig[1];   // rising edge
   #sP_Trig[1] := #ioHMI_Interface.CMD.RequestPB;
   #_w2 := #_w1 AND #iSysInface.ManualMode;
   IF #_w2 AND (NOT #"iSafetyGate Opened Monitor" OR #"iSafetyGate Opened Monitor") AND #ioSafetyGateLock THEN
       #"sSafetyGate UnlockRequest" := TRUE;
       #"sSafetyGate LockRequest" := FALSE;
   END_IF;
   IF #_w2 AND NOT #"iSafetyGate Opened Monitor" AND NOT #ioSafetyGateLock THEN
       #"sSafetyGate LockRequest" := TRUE;
       #"sSafetyGate UnlockRequest" := FALSE;
   END_IF;
END_REGION

REGION Network 4: 安全门开门请求标志位 / Safety door opening request flag bit
   RUNG wire#powerrail
      Contact( #tAlyways_On )
      wire#w1
      I_Contact( #iSysInface.ManualMode )
      { S7_Templates := "SrcType := Int" } NE_Contact(in1 := #iMode, in2 := 2)
      R_Coil( #"sSafetyGate UnlockRequest" )
   END_RUNG
   RUNG wire#w1
      Contact( #iSysInface.ManualMode )
      P_Trig( #sP_Trig[2] )
      wire#w2
      R_Coil( #"sSafetyGate UnlockRequest" )
   END_RUNG
   RUNG wire#w2
      R_Coil( #"sSafetyGate LockRequest" )
   END_RUNG
   RUNG wire#w1
      Contact( #ioSafetyGateLock )
      wire#w3
      N_Trig( #sN_Trig[1] )
      R_Coil( #"sSafetyGate UnlockRequest" )
   END_RUNG
   RUNG wire#w3
      P_Trig( #sP_Trig[3] )
      R_Coil( #"sSafetyGate LockRequest" )
   END_RUNG
   // the same network as SCL:
   IF #tAlyways_On AND NOT #iSysInface.ManualMode AND (#iMode <> 2) THEN
       #"sSafetyGate UnlockRequest" := FALSE;
   END_IF;
   #_w1 := #tAlyways_On AND #iSysInface.ManualMode;
   #_w2 := #_w1 AND NOT #sP_Trig[2];   // rising edge
   #sP_Trig[2] := #_w1;
   IF #_w2 THEN
       #"sSafetyGate UnlockRequest" := FALSE;
       #"sSafetyGate LockRequest" := FALSE;
   END_IF;
   #_w3 := #tAlyways_On AND #ioSafetyGateLock;
   #_w4 := NOT #_w3 AND #sN_Trig[1];   // falling edge
   #sN_Trig[1] := #_w3;
   IF #_w4 THEN #"sSafetyGate UnlockRequest" := FALSE; END_IF;
   #_w5 := #_w3 AND NOT #sP_Trig[3];   // rising edge
   #sP_Trig[3] := #_w3;
   IF #_w5 THEN #"sSafetyGate LockRequest" := FALSE; END_IF;
END_REGION

REGION Network 5: Reset SafetyGateLock
   // 安全门解锁
   RUNG wire#powerrail
      Contact( #iSysInface.ManualMode )
      Contact( #"sSafetyGate UnlockRequest" )
      wire#w1
      I_Contact( #"iSafetyGate Opened Monitor" )
      wire#w2
      R_Coil( #ioSafetyGateLock )
   END_RUNG
   RUNG wire#w1
      Contact( #"iSafetyGate Opened Monitor" )
   END_RUNG wire#w2
   RUNG wire#powerrail
      Contact( #iSysInface.Auto.Mode )
      { S7_Templates := "SrcType := Int" } EQ_Contact(in1 := #iMode, in2 := 2)
      Contact( #"sSafetyGate UnlockRequest" )
   END_RUNG wire#w2
   // the same network as SCL:
   IF (#iSysInface.ManualMode AND #"sSafetyGate UnlockRequest" AND (NOT #"iSafetyGate Opened Monitor" OR #"iSafetyGate Opened Monitor")) OR (#iSysInface.Auto.Mode AND (#iMode = 2) AND #"sSafetyGate UnlockRequest") THEN
       #ioSafetyGateLock := FALSE;
   END_IF;
END_REGION

